//	//If Soft EStop is pressed, turn off 1027, 1028, 1029, 1030, 1031
//	IF KR4_Estop THEN		
//		bOutBit[2,0]:=bOutBit[2,1]:=bOutBit[2,2]:=bOutBit[2,3]:=bOutBit[2,4]:=bOutBit[2,5]:=bOutBit[2,6]:=FALSE;
//	END_IF
	
//	//================================ Function IO
	
//	PLC_O_D2.0 := bOutBit[2,0]; //1027
//	PLC_O_D2.1 := bOutBit[2,1]; //1028
//	PLC_O_D2.2 := bOutBit[2,2]; //1029
//	PLC_O_D2.3 := bOutBit[2,3]; //1030
//	PLC_O_D2.4 := bOutBit[2,4]; //1031
//	PLC_O_D2.5 := bOutBit[2,5]; //1032
//	PLC_O_D2.6 := bOutBit[2,6]; //1033
//	PLC_O_D2.7 := bOutBit[2,7]; //1034
	
//	PLC_O_D3.0 := bOutBit[3,0]; //1035
//	PLC_O_D3.1 := bOutBit[3,1]; //1036
//	PLC_O_D3.2 := bOutBit[3,2]; //1037
//	PLC_O_D3.3 := bOutBit[3,3]; //1038
//	PLC_O_D3.4 := bOutBit[3,4]; //1039
//	PLC_O_D3.5 := bOutBit[3,5]; //1040
//	PLC_O_D3.6 := bOutBit[3,6]; //1041
//	PLC_O_D3.7 := bOutBit[3,7]; //1042
	
//	bInBit[2,0] := PLC_I_D2.0; //993
//	bInBit[2,1] := PLC_I_D2.1; //994
//	bInBit[2,2] := PLC_I_D2.2; //995
//	bInBit[2,3] := PLC_I_D2.3; //996
//	bInBit[2,4] := PLC_I_D2.4; //997
//	bInBit[2,5] := PLC_I_D2.5; //998
//	bInBit[2,6] := PLC_I_D2.6; //999
//	bInBit[2,7] := PLC_I_D2.7; //1000
	
//	bInBit[3,0] := PLC_I_D3.0; //1001
//	bInBit[3,1] := PLC_I_D3.1; //1002
//	bInBit[3,2] := PLC_I_D3.2; //1003
//	bInBit[3,3] := PLC_I_D3.3; //1004
//	bInBit[3,4] := PLC_I_D3.4; //1005
//	bInBit[3,5] := PLC_I_D3.5; //1006
//	bInBit[3,6] := PLC_I_D3.6; //1007
//	bInBit[3,7] := PLC_I_D3.7; //1008

//	//================================ Motion IO
	
//	IF NoMotion THEN
//		RETURN;
//	END_IF
	
//	PLC_O_D1.0 := bOutBit[1,0]; //300
//	PLC_O_D1.1 := bOutBit[1,1]; //301
//	PLC_O_D1.2 := bOutBit[1,2]; //302
//	PLC_O_D1.3 := bOutBit[1,3]; //303
//	PLC_O_D1.4 := bOutBit[1,4]; //304
//	PLC_O_D1.5 := bOutBit[1,5]; //305
//	PLC_O_D1.6 := bOutBit[1,6]; //306
//	PLC_O_D1.7 := bOutBit[1,7]; //307
	
//	bInBit[1,0] := PLC_I_D1.0; //300
//	bInBit[1,1] := PLC_I_D1.1; //301
//	bInBit[1,2] := PLC_I_D1.2; //302
//	bInBit[1,3] := PLC_I_D1.3; //303
//	bInBit[1,4] := PLC_I_D1.4; //304
//	bInBit[1,5] := PLC_I_D1.5; //305
//	bInBit[1,6] := PLC_I_D1.6; //306
//	bInBit[1,7] := PLC_I_D1.7; //307
	
//	IF PLC_I_D1 = 1 THEN
//		Idle := TRUE;
//	ELSE
//		Idle := FALSE;
//	END_IF

END_PROGRAM

// ---- POUs/Kuka IO/KR5.TcPOU
PROGRAM KR5
VAR_INPUT
	PLC_O_SYS 	AT %Q* : DWORD;
	PLC_O_PROG1 AT %Q* : DWORD;
	
	PLC_I_SYS 	AT %I* : DWORD;
	PLC_I_PROG1 AT %I* : DWORD;
	PLC_I_AXIS 	AT %I* : ARRAY[1..6] OF DWORD;
	PLC_I_CURR	AT %I* : ARRAY[1..6] OF DWORD;
	PLC_I_TEMP	AT %I* : ARRAY[1..6] OF DWORD;
	
	KR5_Estop		: BOOL;
	Idle			: BOOL;
	NoMotion		: BOOL;
	
	bOutBit : ARRAY [1..6,0..7] OF BOOL;
	bInBit  : ARRAY [1..6,0..7] OF BOOL;
	index		: USINT;
	index1		: USINT;
	
	dAxis		: ARRAY[1..6] OF DWORD;
	dCurr		: ARRAY[1..6] OF DWORD;
	dTemp		: ARRAY[1..6] OF DWORD;
END_VAR

VAR
	KROnline: BOOL;
	KR_ProgReady: BOOL;
END_VAR

	//If Soft EStop is pressed, turn off 1027 ~ 1034
	IF KR5_Estop THEN		
		bOutBit[1,0]:=bOutBit[1,1]:=bOutBit[1,2]:=bOutBit[1,3]:=
		bOutBit[1,4]:=bOutBit[1,5]:=bOutBit[1,6]:=bOutBit[1,7]:=FALSE;
	END_IF

	//Idle 	
	IF 	PLC_I_PROG1 = 1 THEN
			Idle := TRUE;
	ELSE
			Idle := FALSE;	
	END_IF
	
	//Online
	IF bInBit[1,0] OR bInBit[1,3] THEN
		KROnline := TRUE;
	ELSE
		KROnline := FALSE;
	END_IF

	//Program Ready
	IF bInBit[1,6] AND bInBit[2,4] THEN
		KR_ProgReady := TRUE;
	ELSIF GVL.KR1_bypass THEN
		KR_ProgReady := TRUE;
	ELSE
		KR_ProgReady := FALSE;
	END_IF
	
	
	// ======================================================================== System IO
	// Data In
	FOR index := 0 TO 31 BY 1 DO
		IF index < 8 THEN
			bInBit[1,index] := DWORD_TO_BOOL( SHR(PLC_I_SYS,index) AND 1);
		ELSIF index > 7 AND index < 16 THEN
			bInBit[2,index-8] := DWORD_TO_BOOL( SHR(PLC_I_SYS,index) AND 1);
		END_IF
	END_FOR
	
	// Data Out
	PLC_O_SYS.0 := bOutBit[1,0]; // 1027 move_enable
	PLC_O_SYS.1 := bOutBit[1,1]; // 1028 Drive_off
	PLC_O_SYS.2 := bOutBit[1,2]; // 1029 IO_Activate
	PLC_O_SYS.3 := bOutBit[1,3]; // 1030 Ext_Start
	PLC_O_SYS.4 := bOutBit[1,4]; // 1031 Conf_mess
	PLC_O_SYS.5 := bOutBit[1,5]; // 1032 
	PLC_O_SYS.6 := bOutBit[1,6]; // 1033 Drive_on
	PLC_O_SYS.7 := bOutBit[1,7]; // 1034 Pgno_Fbit
	PLC_O_SYS.8 := bOutBit[2,0]; // 1035 Pgno_Valid
	PLC_O_SYS.9 := bOutBit[2,1]; // 1036 Pgno_Parity

	// ===================================================================== Programme IO
	FOR index := 0 TO 31 BY 1 DO
		IF index < 8 THEN
			bInBit[3,index] := DWORD_TO_BOOL( SHR(PLC_I_PROG1,index) AND 1);
		ELSIF index > 7 AND index < 16 THEN
			bInBit[4,index-8] := DWORD_TO_BOOL( SHR(PLC_I_PROG1,index) AND 1);
		ELSIF index > 15 AND index < 24 THEN
			bInBit[5,index-16] := DWORD_TO_BOOL( SHR(PLC_I_PROG1,index) AND 1);
		ELSIF index > 23 THEN
			bInBit[6,index-24] := DWORD_TO_BOOL( SHR(PLC_I_PROG1,index) AND 1);
		END_IF
	END_FOR
	
	
	PLC_O_PROG1.0 := bOutBit[3,0]; // 200
	PLC_O_PROG1.1 := bOutBit[3,1]; // 201
	PLC_O_PROG1.2 := bOutBit[3,2]; // 202
	PLC_O_PROG1.3 := bOutBit[3,3]; // 203
	PLC_O_PROG1.4 := bOutBit[3,4]; // 204
	PLC_O_PROG1.5 := bOutBit[3,5]; // 205
	PLC_O_PROG1.6 := bOutBit[3,6]; // 206
	PLC_O_PROG1.7 := bOutBit[3,7]; // 207
	PLC_O_PROG1.8 := bOutBit[4,0]; // 208
	PLC_O_PROG1.9 := bOutBit[4,1]; // 209
	PLC_O_PROG1.10 := bOutBit[4,2]; // 210
	PLC_O_PROG1.11 := bOutBit[4,3]; // 211
	PLC_O_PROG1.12 := bOutBit[4,4]; // 212
	PLC_O_PROG1.13 := bOutBit[4,5]; // 213
	PLC_O_PROG1.14 := bOutBit[4,6]; // 214
	PLC_O_PROG1.15 := bOutBit[4,7]; // 215
	PLC_O_PROG1.16 := bOutBit[5,0]; // 216
	PLC_O_PROG1.17 := bOutBit[5,1]; // 217
	PLC_O_PROG1.18 := bOutBit[5,2]; // 218
	PLC_O_PROG1.19 := bOutBit[5,3]; // 219
	PLC_O_PROG1.20 := bOutBit[5,4]; // 220
	PLC_O_PROG1.21 := bOutBit[5,5]; // 221
	PLC_O_PROG1.22 := bOutBit[5,6]; // 222
	PLC_O_PROG1.23 := bOutBit[5,7]; // 223
	PLC_O_PROG1.24 := bOutBit[6,0]; // 224
	PLC_O_PROG1.25 := bOutBit[6,1]; // 225
	PLC_O_PROG1.26 := bOutBit[6,2]; // 226
	PLC_O_PROG1.27 := bOutBit[6,3]; // 227
	PLC_O_PROG1.28 := bOutBit[6,4]; // 228
	PLC_O_PROG1.29 := bOutBit[6,5]; // 229
	PLC_O_PROG1.30 := bOutBit[6,6]; // 230
	PLC_O_PROG1.31 := bOutBit[6,7]; // 231
	
	// ===================================================================== Robot Data
	FOR index1 := 1 TO 6 BY 1 DO
		FOR index := 0 TO 31 BY 1 DO
			dAxis[index1] := PLC_I_AXIS[index1];
			dCurr[index1] := PLC_I_CURR[index1];
			dTemp[index1] := PLC_I_TEMP[index1];
		END_FOR
	END_FOR
	
	
	
	
	
	
	
	
	
//	//================================ Function IO
	
//	PLC_O_D1.0 := bOutBit[1,0]; //1027 motion enable (on to start motor)
//	PLC_O_D1.1 := bOutBit[1,1]; //1028 Drives off (inverse) (on to start motor)
//	PLC_O_D1.2 := bOutBit[1,2]; //1029 Activate interface (on to start motor)
//	PLC_O_D1.3 := bOutBit[1,3]; //1030 Prog Start
//	PLC_O_D1.4 := bOutBit[1,4]; //1031 Acknowledge error msg
//	PLC_O_D1.5 := bOutBit[1,5]; //1032 Drives on
//	PLC_O_D1.6 := bOutBit[1,6]; //1033
//	PLC_O_D1.7 := bOutBit[1,7]; //1034
	
//	PLC_O_D2.0 := bOutBit[2,0]; //1035
//	PLC_O_D2.1 := bOutBit[2,1]; //1036
//	PLC_O_D2.2 := bOutBit[2,2]; //1037
//	PLC_O_D2.3 := bOutBit[2,3]; //1038
//	PLC_O_D2.4 := bOutBit[2,4]; //1039
//	PLC_O_D2.5 := bOutBit[2,5]; //1040
//	PLC_O_D2.6 := bOutBit[2,6]; //1041
//	PLC_O_D2.7 := bOutBit[2,7]; //1042
	
//	bInBit[1,0] := PLC_I_D1.0; //993
//	bInBit[1,1] := PLC_I_D1.1; //994
//	bInBit[1,2] := PLC_I_D1.2; //995
//	bInBit[1,3] := PLC_I_D1.3; //996
//	bInBit[1,4] := PLC_I_D1.4; //997
//	bInBit[1,5] := PLC_I_D1.5; //998
//	bInBit[1,6] := PLC_I_D1.6; //999
//	bInBit[1,7] := PLC_I_D1.7; //1000
	
//	bInBit[2,0] := PLC_I_D2.0; //1001
//	bInBit[2,1] := PLC_I_D2.1; //1002
//	bInBit[2,2] := PLC_I_D2.2; //1003
//	bInBit[2,3] := PLC_I_D2.3; //1004
//	bInBit[2,4] := PLC_I_D2.4; //1005
//	bInBit[2,5] := PLC_I_D2.5; //1006
//	bInBit[2,6] := PLC_I_D2.6; //1007
//	bInBit[2,7] := PLC_I_D2.7; //1008
	
//	//================================ Motion IO
	
//	IF NoMotion THEN
//		RETURN;
//	END_IF
	
//	PLC_O_D3.0 := bOutBit[3,0]; //200
//	PLC_O_D3.1 := bOutBit[3,1]; //201
//	PLC_O_D3.2 := bOutBit[3,2]; //202
//	PLC_O_D3.3 := bOutBit[3,3]; //203
//	PLC_O_D3.4 := bOutBit[3,4]; //204
//	PLC_O_D3.5 := bOutBit[3,5]; //205
//	PLC_O_D3.6 := bOutBit[3,6]; //206
//	PLC_O_D3.7 := bOutBit[3,7]; //207
	
//	PLC_O_D4.0 := bOutBit[4,0]; //208
//	PLC_O_D4.1 := bOutBit[4,1]; //209
//	PLC_O_D4.2 := bOutBit[4,2]; //210
//	PLC_O_D4.3 := bOutBit[4,3]; //211
//	PLC_O_D4.4 := bOutBit[4,4]; //212
//	PLC_O_D4.5 := bOutBit[4,5]; //213
//	PLC_O_D4.6 := bOutBit[4,6]; //214
//	PLC_O_D4.7 := bOutBit[4,7]; //215
	
//	PLC_O_D5.0 := bOutBit[5,0]; //216
//	PLC_O_D5.1 := bOutBit[5,1]; //217
//	PLC_O_D5.2 := bOutBit[5,2]; //218
//	PLC_O_D5.3 := bOutBit[5,3]; //219
//	PLC_O_D5.4 := bOutBit[5,4]; //220
//	PLC_O_D5.5 := bOutBit[5,5]; //221
//	PLC_O_D5.6 := bOutBit[5,6]; //222
//	PLC_O_D5.7 := bOutBit[5,7]; //223

//	PLC_O_D6.0 := bOutBit[6,0]; //224
//	PLC_O_D6.1 := bOutBit[6,1]; //225
//	PLC_O_D6.2 := bOutBit[6,2]; //226
//	PLC_O_D6.3 := bOutBit[6,3]; //227
//	PLC_O_D6.4 := bOutBit[6,4]; //228
//	PLC_O_D6.5 := bOutBit[6,5]; //229
//	PLC_O_D6.6 := bOutBit[6,6]; //230
//	PLC_O_D6.7 := bOutBit[6,7]; //231

//	bInBit[3,0] := PLC_I_D3.0; //200
//	bInBit[3,1] := PLC_I_D3.1; //201
//	bInBit[3,2] := PLC_I_D3.2; //202
//	bInBit[3,3] := PLC_I_D3.3; //203
//	bInBit[3,4] := PLC_I_D3.4; //204
//	bInBit[3,5] := PLC_I_D3.5; //205
//	bInBit[3,6] := PLC_I_D3.6; //206
//	bInBit[3,7] := PLC_I_D3.7; //207
	
//	bInBit[4,0] := PLC_I_D4.0; //208
//	bInBit[4,1] := PLC_I_D4.1; //209
//	bInBit[4,2] := PLC_I_D4.2; //210
//	bInBit[4,3] := PLC_I_D4.3; //211
//	bInBit[4,4] := PLC_I_D4.4; //212
//	bInBit[4,5] := PLC_I_D4.5; //213
//	bInBit[4,6] := PLC_I_D4.6; //214
//	bInBit[4,7] := PLC_I_D4.7; //215
	
//	bInBit[5,0] := PLC_I_D5.0; //216
//	bInBit[5,1] := PLC_I_D5.1; //217
//	bInBit[5,2] := PLC_I_D5.2; //218
//	bInBit[5,3] := PLC_I_D5.3; //219
//	bInBit[5,4] := PLC_I_D5.4; //220
//	bInBit[5,5] := PLC_I_D5.5; //221
//	bInBit[5,6] := PLC_I_D5.6; //222
//	bInBit[5,7] := PLC_I_D5.7; //223
	
//	bInBit[6,0] := PLC_I_D6.0; //224
//	bInBit[6,1] := PLC_I_D6.1; //225
//	bInBit[6,2] := PLC_I_D6.2; //226
//	bInBit[6,3] := PLC_I_D6.3; //227
//	bInBit[6,4] := PLC_I_D6.4; //228
//	bInBit[6,5] := PLC_I_D6.5; //229
//	bInBit[6,6] := PLC_I_D6.6; //230
//	bInBit[6,7] := PLC_I_D6.7; //231
	
	
	
//	//If Soft EStop is pressed, turn off 1027, 1028, 1029, 1030, 1031
//	IF KR5_Estop THEN		
//		bOutBit[3,0]:=bOutBit[3,1]:=bOutBit[3,2]:=bOutBit[3,3]:=bOutBit[3,4]:=bOutBit[2,5]:=bOutBit[2,6]:=FALSE;
//	END_IF
	
//	//================================ Function IO
	
//	PLC_O_D3.0 := bOutBit[3,0]; //1027
//	PLC_O_D3.1 := bOutBit[3,1]; //1028
//	PLC_O_D3.2 := bOutBit[3,2]; //1029
//	PLC_O_D3.3 := bOutBit[3,3]; //1030
//	PLC_O_D3.4 := bOutBit[3,4]; //1031
//	PLC_O_D3.5 := bOutBit[3,5]; //1032
//	PLC_O_D3.6 := bOutBit[3,6]; //1033
//	PLC_O_D3.7 := bOutBit[3,7]; //1034
	
//	PLC_O_D4.0 := bOutBit[4,0]; //1035
//	PLC_O_D4.1 := bOutBit[4,1]; //1036
//	PLC_O_D4.2 := bOutBit[4,2]; //1037
//	PLC_O_D4.3 := bOutBit[4,3]; //1038
//	PLC_O_D4.4 := bOutBit[4,4]; //1039
//	PLC_O_D4.5 := bOutBit[4,5]; //1040
//	PLC_O_D4.6 := bOutBit[4,6]; //1041
//	PLC_O_D4.7 := bOutBit[4,7]; //1042
	
//	bInBit[3,0] := PLC_I_D3.0; //993
//	bInBit[3,1] := PLC_I_D3.1; //994
//	bInBit[3,2] := PLC_I_D3.2; //995
//	bInBit[3,3] := PLC_I_D3.3; //996
//	bInBit[3,4] := PLC_I_D3.4; //997
//	bInBit[3,5] := PLC_I_D3.5; //998
//	bInBit[3,6] := PLC_I_D3.6; //999
//	bInBit[3,7] := PLC_I_D3.7; //1000
	
//	bInBit[4,0] := PLC_I_D4.0; //1001
//	bInBit[4,1] := PLC_I_D4.1; //1002
//	bInBit[4,2] := PLC_I_D4.2; //1003
//	bInBit[4,3] := PLC_I_D4.3; //1004
//	bInBit[4,4] := PLC_I_D4.4; //1005
//	bInBit[4,5] := PLC_I_D4.5; //1006
//	bInBit[4,6] := PLC_I_D4.6; //1007
//	bInBit[4,7] := PLC_I_D4.7; //1008
	
//	//================================ Motion IO
	
//	IF NoMotion THEN
//		RETURN;
//	END_IF

//	PLC_O_D1.0 := bOutBit[1,0]; //200
//	PLC_O_D1.1 := bOutBit[1,1]; //201
//	PLC_O_D1.2 := bOutBit[1,2]; //202
//	PLC_O_D1.3 := bOutBit[1,3]; //203
//	PLC_O_D1.4 := bOutBit[1,4]; //204
//	PLC_O_D1.5 := bOutBit[1,5]; //205
//	PLC_O_D1.6 := bOutBit[1,6]; //206
//	PLC_O_D1.7 := bOutBit[1,7]; //207
	
//	PLC_O_D2.0 := bOutBit[2,0]; //208
//	PLC_O_D2.1 := bOutBit[2,1]; //209
//	PLC_O_D2.2 := bOutBit[2,2]; //210
//	PLC_O_D2.3 := bOutBit[2,3]; //211
//	PLC_O_D2.4 := bOutBit[2,4]; //212
//	PLC_O_D2.5 := bOutBit[2,5]; //213
//	PLC_O_D2.6 := bOutBit[2,6]; //214
//	PLC_O_D2.7 := bOutBit[2,7]; //215
	
//	bInBit[1,0] := PLC_I_D1.0; //200
//	bInBit[1,1] := PLC_I_D1.1; //201
//	bInBit[1,2] := PLC_I_D1.2; //202
//	bInBit[1,3] := PLC_I_D1.3; //203
//	bInBit[1,4] := PLC_I_D1.4; //204
//	bInBit[1,5] := PLC_I_D1.5; //205
//	bInBit[1,6] := PLC_I_D1.6; //206
//	bInBit[1,7] := PLC_I_D1.7; //207
	
//	bInBit[2,0] := PLC_I_D2.0; //208
//	bInBit[2,1] := PLC_I_D2.1; //209
//	bInBit[2,2] := PLC_I_D2.2; //210
//	bInBit[2,3] := PLC_I_D2.3; //211
//	bInBit[2,4] := PLC_I_D2.4; //212
//	bInBit[2,5] := PLC_I_D2.5; //213
//	bInBit[2,6] := PLC_I_D2.6; //214
//	bInBit[2,7] := PLC_I_D2.7; //215

//	IF PLC_I_D1 = 1 THEN
//		Idle := TRUE;
//	ELSE
//		Idle := FALSE;
//	END_IF

END_PROGRAM

// ---- POUs/RESET_SEQ.TcPOU
PROGRAM RESET_SEQ
VAR_INPUT
	Reset_seq	: INT;
	log_reset	: STRING[255];
END_VAR
VAR
	RstTON		: TON;
	RstToff		: TON;
	bOn			: BOOL;
	bLastOn		: BOOL;
	Bit1		: INT;
	Bit2		: INT;
END_VAR


	//Off time
	RstTON(IN:= NOT RstTOff.Q, PT:= T#0.2S, Q=> bOn , ET=> );
	//On time
	RstTOff(IN:= bOn, PT:= T#0.5S, Q=> , ET=> );
	
	IF bOn <> bLastOn THEN
		IF bON THEN
			IF Reset_seq < 14 THEN
				IF Reset_seq =2 THEN
					IF KR1.bInBit[1,6] AND KR2.bInBit[1,6] AND KR3.bInBit[1,6] AND KR4.bInBit[1,6] AND KR5.bInBit[1,6] THEN
						Reset_seq := Reset_seq + 1;	
					END_IF
				ELSE	
					Reset_seq := Reset_seq + 1;
				END_IF			
			ELSE
				Reset_seq 	:=0;
				bOn 		:= FALSE;
			END_IF
		END_IF
	END_IF
	
	CASE Reset_seq OF
		0:
			IF NOT GVL.KR1_bypass THEN
				FOR Bit1 := 1 TO 30 BY 1 DO
					FOR Bit2 := 0 TO 7 BY 1 DO
						KR1.bOutBit[Bit1,Bit2] := FALSE;
					END_FOR
				END_FOR
			END_IF
			IF NOT GVL.KR2_bypass THEN
				FOR Bit1 := 1 TO 8 BY 1 DO
					FOR Bit2 := 0 TO 7 BY 1 DO
						KR2.bOutBit[Bit1,Bit2] := FALSE;
					END_FOR
				END_FOR
			END_IF
			IF NOT GVL.KR3_bypass THEN
				FOR Bit1 := 1 TO 3 BY 1 DO
					FOR Bit2 := 0 TO 7 BY 1 DO
						KR3.bOutBit[Bit1,Bit2] := FALSE;
					END_FOR
				END_FOR
			END_IF
			IF NOT GVL.KR4_bypass THEN
				FOR Bit1 := 1 TO 3 BY 1 DO
					FOR Bit2 := 0 TO 7 BY 1 DO
						KR4.bOutBit[Bit1,Bit2] := FALSE;
					END_FOR
				END_FOR
			END_IF
			IF NOT GVL.KR5_bypass THEN
				FOR Bit1 := 1 TO 6 BY 1 DO
					FOR Bit2 := 0 TO 7 BY 1 DO
						KR5.bOutBit[Bit1,Bit2] := FALSE;
					END_FOR
				END_FOR
			END_IF
		1:
			IF NOT GVL.KR1_bypass THEN
				KR1.bOutBit[1,0]:=KR1.bOutBit[1,1]:=KR1.bOutBit[1,2]:=TRUE;
			END_IF
			IF NOT GVL.KR2_bypass THEN
				KR2.bOutBit[1,0]:=KR2.bOutBit[1,1]:=KR2.bOutBit[1,2]:=TRUE;
			END_IF
			IF NOT GVL.KR3_bypass THEN
				KR3.bOutBit[1,0]:=KR3.bOutBit[1,1]:=KR3.bOutBit[1,2]:=TRUE;
			END_IF
			IF NOT GVL.KR4_bypass THEN
				KR4.bOutBit[1,0]:=KR4.bOutBit[1,1]:=KR4.bOutBit[1,2]:=TRUE;
			END_IF
			IF NOT GVL.KR5_bypass THEN
				KR5.bOutBit[1,0]:=KR5.bOutBit[1,1]:=KR5.bOutBit[1,2]:=TRUE;
			END_IF
		2:
			IF NOT GVL.KR1_bypass THEN
				KR1.bOutBit[1,4] := TRUE; //1031
			END_IF
			IF NOT GVL.KR2_bypass THEN
				KR2.bOutBit[1,4] := TRUE; //1031
			END_IF
			IF NOT GVL.KR3_bypass THEN
				KR3.bOutBit[1,4] := TRUE; //1031
			END_IF
			IF NOT GVL.KR4_bypass THEN
				KR4.bOutBit[1,4] := TRUE; //1031
			END_IF
			IF NOT GVL.KR5_bypass THEN
				KR5.bOutBit[1,4] := TRUE; //1031
			END_IF
		3:
			IF NOT GVL.KR1_bypass THEN
				KR1.bOutBit[1,4] := FALSE; //1031
			END_IF
			IF NOT GVL.KR2_bypass THEN
				KR2.bOutBit[1,4] := FALSE; //1031
			END_IF
			IF NOT GVL.KR3_bypass THEN
				KR3.bOutBit[1,4] := FALSE; //1031
			END_IF
			IF NOT GVL.KR4_bypass THEN
				KR4.bOutBit[1,4] := FALSE; //1031
			END_IF
			IF NOT GVL.KR5_bypass THEN
				KR5.bOutBit[1,4] := FALSE; //1031
			END_IF
		4:
			KR1.bOutBit[1,5] := TRUE; //1032
		5:
			KR2.bOutBit[1,6] := TRUE; //1033
		6:
			KR3.bOutBit[1,5] := TRUE; //1032
		7:	
			KR4.bOutBit[1,5] := TRUE; //1032
		8:		
			KR5.bOutBit[1,5] := TRUE; //1032
		9:
			KR1.bOutBit[1,5] := FALSE; //1032
			KR1.bOutBit[1,3] := TRUE; //1030
		10:
			KR2.bOutBit[1,6] := FALSE; //1033
			KR2.bOutBit[1,3] := TRUE; //1030
		11:
			KR3.bOutBit[1,5] := FALSE; //1032
			KR3.bOutBit[1,3] := TRUE; //1030
		12:
			KR4.bOutBit[1,5] := FALSE; //1032
			KR4.bOutBit[1,3] := TRUE; //1030
		13:
			KR5.bOutBit[1,5] := FALSE; //1032
			KR5.bOutBit[1,3] := TRUE; //1030
		14:
			AUTO_MODE.Halt_Production := FALSE;
			Reset_seq :=0;
			MAIN.Reset_State := FALSE;
			MAIN.btn_Reset := FALSE;
	END_CASE
	bLastOn := bOn;

END_PROGRAM

// ---- POUs/Auto_Seq/AUTO_MODE.TcPOU
PROGRAM AUTO_MODE
VAR_INPUT
	Reset_seq_btn	: BOOL;
	Start_time	: string;
	
	JIGA_WELDING: BOOL;
	JIGB_WELDING: BOOL;
	JIGC_WELDING: BOOL;
	TT_WELDING	: BOOL;
	IF_PICK		: BOOL;
	JIGC_PICK	: BOOL;
	VB_PICK		: BOOL;
	
	JIGA_LOAD	: BOOL;
	JIGB_LOAD	: BOOL;
	JIGC_LOAD	: BOOL;
	TT_LOAD		: BOOL;
	CR_PICK		: BOOL;
	
	AutoMode	: BOOL;
	ManualMode	: BOOL;
	next_step	: BOOL;
	Halt_Production	: BOOL;
	
	processnameA5 : STRING[255];
	processnameA4 : STRING[255];
	processnameA3 : STRING[255];
	processnameA2 : STRING[255];
	processnameA1 : STRING[255];
	processnameCR : STRING[255];
	processnameRW : STRING[255];
	processnameFG : STRING[255];
	processnameCOSMO : STRING[255];
	
	COSMO_LOAD	: BOOL;
	COSMO_RUN	: BOOL;
	CR_UNLOADING: BOOL;
	
	CLEAR_COSMO	: Bool;
	KR1_PITSTOP : BOOL;
	FG_PACKING	: BOOL;
	RW_PACKING	: BOOL;
	
	A4_Run_Flag : BOOL;
	A3_Run_Flag : BOOL;
	A2_Run_Flag : BOOL;
	A1_Run_Flag : BOOL;
	
	Run_Next_Rack : BOOL:= TRUE;
	Out_time	: STRING;
	JIGA_ErrorState : BOOL;
	JIGB_ErrorState : BOOL;
	JIGC_ErrorState : BOOL;
	TT_ErrorState 	: BOOL;
END_VAR
VAR
	Auto_IntOn	: TON;
	Auto_IntOff	: TON;
	Auto_on		: BOOL;
	Auto_laston	: BOOL;
	
	Bit1: INT;
	Bit2: INT;
END_VAR

IF next_step OR Automode THEN
	IF NOT KR2.KR_ProgReady OR NOT KR3.KR_ProgReady OR NOT KR4.KR_ProgReady OR NOT KR5.KR_ProgReady THEN
		Automode := FALSE;
	END_IF
	IF_RACK_CHECK();
	SEQ_A5();
	SEQ_A4();
	SEQ_A3();
	SEQ_A2();
	SEQ_A1();
	SEQ_B5();
	SEQ_B4();
	SEQ_B3();
	SEQ_B2();
	SEQ_B1();
		
	SEQ_CR_PICK();
//	SEQ_LP_LYR0();
	SEQ_FG_A();
	SEQ_COSMO();
	
	 
END_IF




IF Reset_seq_btn THEN
	
	
	IF_RACK_CHECK.checkIn_A5 := IF_RACK_CHECK.checkIn_A4 := IF_RACK_CHECK.checkIn_A3 := IF_RACK_CHECK.checkIn_A2 := IF_RACK_CHECK.checkIn_A1 := 
	IF_RACK_CHECK.checkIn_B5 := IF_RACK_CHECK.checkIn_B4 := IF_RACK_CHECK.checkIn_B3 := IF_RACK_CHECK.checkIn_B2 := IF_RACK_CHECK.checkIn_B1 := FALSE;
	
	SEQ_A5.A5_sequence		:= SEQ_A4.A4_sequence		:= SEQ_A3.A3_sequence	:= SEQ_A2.A2_sequence	:= SEQ_A1.A1_sequence:=
	SEQ_B5.B5_sequence		:= SEQ_B4.B4_sequence		:= SEQ_B3.B3_sequence	:= SEQ_B2.B2_sequence	:= SEQ_B1.B1_sequence:=
	SEQ_CR_PICK.CR_sequence	:= SEQ_COSMO.COSMO_sequence	:= SEQ_RW.RW_sequence 	:= SEQ_FG_A.FG_sequence	:= SEQ_LYR_PD0.LYRPD_sequence := 0;
	
	processnameA5 := processnameA4 := processnameA3 := processnameA2 	:= processnameA1 :=
	processnameCR := processnameRW := processnameFG := processnameCOSMO := '';  
	
	IF_PICK			:= JIGC_PICK		:= CR_PICK			:=
	JIGA_WELDING 	:= JIGB_WELDING 	:= JIGC_WELDING		:= TT_WELDING   	:= 
	JIGA_LOAD 	 	:= JIGB_LOAD  	 	:= JIGC_LOAD 		:= TT_LOAD			:=
	GVL.JIGA_Clamp 	:= GVL.JIGB_Clamp 	:= GVL.JIGC_Clamp 	:= CR_UNLOADING	 	:= 
	COSMO_LOAD 	 	:= COSMO_RUN 	 	:= CLEAR_COSMO  	:= KR1_PITSTOP 		:= 
	FG_PACKING 	 	:= RW_PACKING 		:= GVL.COSMO_Run	:= GVL.TTorch_Run 	:= FALSE;
	
	JIGA_ErrorState := JIGB_ErrorState 	:= JIGC_ErrorState 	:= TT_ErrorState 	:= FALSE;
	Automode 		:= next_step 		:= FALSE;
	Run_Next_Rack 	:= TRUE;
	Halt_Production := FALSE;
	
	GVL.Layerpad := FALSE;
	GVL.COSMO_UNLOAD := FALSE;

	FOR Bit1 := 2 TO 30 BY 1 DO
		FOR Bit2 := 0 TO 7 BY 1 DO
			KR1.bOutBit[Bit1,Bit2] := FALSE;
		END_FOR
	END_FOR
	FOR Bit1 := 2 TO 8 BY 1 DO
		FOR Bit2 := 0 TO 7 BY 1 DO
			KR2.bOutBit[Bit1,Bit2] := FALSE;
		END_FOR
	END_FOR
	FOR Bit1 := 2 TO 3 BY 1 DO
		FOR Bit2 := 0 TO 7 BY 1 DO
			KR3.bOutBit[Bit1,Bit2] := FALSE;
			KR4.bOutBit[Bit1,Bit2] := FALSE;
		END_FOR
	END_FOR
	FOR Bit1 := 2 TO 6 BY 1 DO
		FOR Bit2 := 0 TO 7 BY 1 DO
			KR5.bOutBit[Bit1,Bit2] := FALSE;
		END_FOR
	END_FOR
	
	Reset_seq_btn := False;
END_IF

END_PROGRAM

// ---- POUs/Auto_Seq/IF_RACK_CHECK.TcPOU
PROGRAM IF_RACK_CHECK
VAR_INPUT
	checkIn_A5 : BOOL;
	checkIn_A4 : BOOL;
	checkIn_A3 : BOOL;
	checkIn_A2 : BOOL;
	checkIn_A1 : BOOL;
	checkIn_B5 : BOOL;
	checkIn_B4 : BOOL;
	checkIn_B3 : BOOL;
	checkIn_B2 : BOOL;
	checkIn_B1 : BOOL;
END_VAR
VAR
	infeedRack_A_empty: BOOL;
	infeedRack_B_empty: BOOL;
	turnflag: BOOL;
	turningA: BOOL;
	turningB: BOOL;
	cool_rack_check : UINT;
END_VAR


IF NOT AUTO_MODE.Run_Next_Rack THEN
	RETURN;
END_IF
	
IF COOL_RACK.CR_full THEN
	RETURN;
END_IF

IF INFEED_RACK.FaceA_InWC THEN
	IF INFEED_RACK.A5_Sensor THEN
		checkIn_A5 := TRUE; AUTO_MODE.Run_Next_Rack := FALSE;
	ELSIF INFEED_RACK.A4_Sensor THEN
		checkIn_A4 := TRUE; AUTO_MODE.Run_Next_Rack := FALSE;
	ELSIF INFEED_RACK.A3_Sensor THEN
		checkIn_A3 := TRUE; AUTO_MODE.Run_Next_Rack := FALSE;
	ELSIF INFEED_RACK.A2_Sensor THEN
		checkIn_A2 := TRUE; AUTO_MODE.Run_Next_Rack := FALSE;
	ELSIF INFEED_RACK.A1_Sensor THEN
		checkIn_A1 := TRUE; AUTO_MODE.Run_Next_Rack := FALSE;
	ELSE
		infeedRack_A_empty := TRUE;	
	END_IF
	
ELSIF INFEED_RACK.FaceB_InWC THEN
	IF INFEED_RACK.B5_Sensor THEN
		checkIn_B5 := TRUE; AUTO_MODE.Run_Next_Rack := FALSE;
	ELSIF INFEED_RACK.B4_Sensor THEN
		checkIn_B4 := TRUE; AUTO_MODE.Run_Next_Rack := FALSE;
	ELSIF INFEED_RACK.B3_Sensor THEN
		checkIn_B3 := TRUE; AUTO_MODE.Run_Next_Rack := FALSE;
	ELSIF INFEED_RACK.B2_Sensor THEN
		checkIn_B2 := TRUE; AUTO_MODE.Run_Next_Rack := FALSE;
	ELSIF INFEED_RACK.B1_Sensor THEN
		checkIn_B1 := TRUE; AUTO_MODE.Run_Next_Rack := FALSE;
	ELSE
		infeedRack_B_empty := TRUE;	
	END_IF
END_IF

IF INFEED_RACK.IFRack_Ready and INFEED_RACK.IFRack_TurnReady THEN
	IF infeedRack_A_empty AND NOT turningB THEN
		turningA := TRUE;
		INFEED_RACK.IFRack_arr[1].5 := FALSE; //BtoA
		INFEED_RACK.IFRack_arr[1].4 := TRUE; //AtoB
		INFEED_RACK(bStart_Write:=TRUE);
		IF INFEED_RACK.FaceB_InWC THEN
			turningA := FALSE;
			infeedRack_A_empty := FALSE;
			INFEED_RACK(bStart_Write:=FALSE);
		END_IF
	ELSIF infeedRack_B_empty AND NOT turningA THEN
		turningB := TRUE;
		INFEED_RACK.IFRack_arr[1].4 := FALSE; //AtoB
		INFEED_RACK.IFRack_arr[1].5 := TRUE; //BtoA
		INFEED_RACK(bStart_Write:=TRUE);
		IF INFEED_RACK.FaceA_InWC THEN
			turningB := FALSE;
			infeedRack_B_empty := FALSE;
			INFEED_RACK(bStart_Write:=FALSE);
		END_IF
	END_IF
END_IF

//INFEED_RACK.bStart_Read:=FALSE;
//INFEED_RACK.bStart_Write:=FALSE;

END_PROGRAM

// ---- POUs/COOL_RACK.TcPOU
PROGRAM COOL_RACK
VAR_INPUT
	bstart_Read		: BOOL;
	bstart_Write	: BOOL;
	iCooling_Time	: INT;
	set_time		: bool;
END_VAR
VAR_OUTPUT
	CR_full 	: bool;
END_VAR
VAR
	WriteCoil	: FB_MBWriteCoils;
	Read_Coils	: FB_MBReadCoils;
	ReadInput: FB_MBReadInputs;
	
	IP_Address		: STRING:='169.254.106.102';
	MB_Port			: UINT	:=502;
	nUnit			: BYTE	:=255; 
	nQuantity		: WORD	:=24;
	nMBAddr			: WORD	:=2048;
	bError_Read		: BOOL;
	bError_Write	: BOOL;
	nErrId_Read		: UDINT;
	nErrId_Write	: UDINT;
	
	CoolRack_arr		: ARRAY [0..2] OF BYTE;

	
	CR	: ARRAY [1..21] OF BOOL;
	num	: INT;
	
	CR_Reset		: INT;
	CR_Sel			: INT;
	CRON			: BOOL;
	CRONlast		: BOOL;
	CRcounterON 	: TON;
	CRcounterOFF	: TON;

END_VAR


//Off time
CRcounterON(IN:= NOT CRcounterOFF.Q, PT:= T#1S, Q=> CRON , ET=> );
//On time
CRcounterOFF(IN:= CRON, PT:= T#1S, Q=> , ET=> );
	
IF CRON <> CRONlast THEN
	FOR CR_Sel := 1 TO 21 BY 1 DO
		IF CR[CR_Sel] THEN
			GVL.CRTimer[CR_Sel] := GVL.CRTimer[CR_Sel] - 1;
		END_IF
	END_FOR
END_IF
CRONlast := CRON;
//================================ Function Block

Read_Coils(
	sIPAddr:= IP_Address, 
	nTCPPort:= MB_Port, 
	nUnitID:= nUnit, 
	nQuantity:= nQuantity, 
	nMBAddr:= nMBAddr, 
	cbLength:= SIZEOF(CoolRack_arr), 
	pDestAddr:= ADR(CoolRack_arr), 
	bExecute:= bstart_Read, 
	tTimeout:= T#1S, 
	bBusy=> , 
	bError=> bError_Read, 
	nErrId=> nErrId_Read, 
	cbRead=> );

WriteCoil(
	sIPAddr:= IP_Address, 
	nTCPPort:= MB_Port, 
	nUnitID:= nUnit, 
	nQuantity:= nQuantity, 
	nMBAddr:= nMBAddr, 
	cbLength:= SIZEOF(CoolRack_arr),  
	pSrcAddr:= ADR(CoolRack_arr), 
	bExecute:= bstart_Write, 
	tTimeout:= T#1S, 
	bBusy=> , 
	bError=> bError_Write, 
	nErrId=> nErrId_Write);

IF set_time THEN
	FOR CR_Reset := 1 TO 21 BY 1 DO
		GVL.CRTimer[CR_Reset] := GVL.iCooling_Time;
	END_FOR	
END_IF

//================================ Sensor

CR[1] := CoolRack_arr[0].0;
CR[2] := CoolRack_arr[0].1;
CR[3] := CoolRack_arr[0].2;
CR[4] := CoolRack_arr[0].3;
CR[5] := CoolRack_arr[0].4;
CR[6] := CoolRack_arr[0].5;
CR[7] := CoolRack_arr[0].6;

CR[8] := CoolRack_arr[0].7;
CR[9] := CoolRack_arr[1].0;
CR[10] := CoolRack_arr[1].1;
CR[11] := CoolRack_arr[1].2;
CR[12] := CoolRack_arr[1].3;
CR[13] := CoolRack_arr[1].4;
CR[14] := CoolRack_arr[1].5;

CR[15] := CoolRack_arr[1].6;
CR[16] := CoolRack_arr[1].7;
CR[17] := CoolRack_arr[2].0;
CR[18] := CoolRack_arr[2].1;
CR[19] := CoolRack_arr[2].2;
CR[20] := CoolRack_arr[2].3;
CR[21] := CoolRack_arr[2].4;

CR[8]:=TRUE;
CR[14]:=TRUE;
CR[15]:=TRUE;
CR[16]:=TRUE;
CR[17]:=TRUE;
CR[18]:=TRUE;
CR[19]:=TRUE;
CR[20]:=TRUE;
CR[21]:=TRUE;
//================================ Cooling Time
FOR num:=1 TO 21 BY 1 DO
	IF NOT CR[num] THEN
		GVL.CRTimer[num] := GVL.iCooling_Time;
	END_IF
//	IF num > 21 THEN
//		num := 1;			
//	END_IF
END_FOR

IF CoolRack_arr[0] = 255 AND CoolRack_arr[1] = 255 AND CoolRack_arr[2] = 31 THEN
	CR_full := TRUE;
ELSE
	CR_full := false;
END_IF

END_PROGRAM

// ---- POUs/INFEED_RACK.TcPOU
PROGRAM INFEED_RACK
VAR_INPUT
	bstart_Read		: BOOL;
	bstart_Write	: BOOL;
	A1_Valve		: BOOL;
	A2_Valve		: BOOL;
	A3_Valve		: BOOL;
	A4_Valve		: BOOL;
	A5_Valve		: BOOL;
	B1_Valve		: BOOL;
	B2_Valve		: BOOL;
	B3_Valve		: BOOL;
	B4_Valve		: BOOL;
	B5_Valve		: BOOL;
	IFRack_Connect	: BOOL;
	IFRack_Ready	: BOOL;
	Turn_A_to_B		: BOOL;
	Turn_B_to_A		: BOOL;
	A1_Sensor		: BOOL;
	A2_Sensor		: BOOL;
	A3_Sensor		: BOOL;
	A4_Sensor		: BOOL;
	A5_Sensor		: BOOL;
	B1_Sensor		: BOOL;
	B2_Sensor		: BOOL;
	B3_Sensor		: BOOL;
	B4_Sensor		: BOOL;
	B5_Sensor		: BOOL;
	FaceA_InWC		: BOOL;
	FaceB_InWC		: BOOL;
	IFRack_TurnReady : BOOL;
	
	IFRack_arr		: ARRAY [0..6] OF BYTE;
END_VAR
VAR
	WriteCoil	: FB_MBWriteCoils;
	Read_Coils	: FB_MBReadCoils;
	ReadInput: FB_MBReadInputs;
	
	IP_Address		: STRING:='169.254.106.101';
	MB_Port			: UINT	:=502;
	nUnit			: BYTE	:=255; 
	nQuantity		: WORD	:=48;
	nMBAddr			: WORD	:=2048;
	bError_Read		: BOOL;
	bError_Write	: BOOL;
	nErrId_Read		: UDINT;
	nErrId_Write	: UDINT;
	
END_VAR


//================================ Function Block

Read_Coils(
	sIPAddr:= IP_Address, 
	nTCPPort:= MB_Port, 
	nUnitID:= nUnit, 
	nQuantity:= nQuantity, 
	nMBAddr:= nMBAddr, 
	cbLength:= SIZEOF(IFRack_arr), 
	pDestAddr:= ADR(IFRack_arr), 
	bExecute:= bstart_Read, 
	tTimeout:= T#1S, 
	bBusy=> , 
	bError=> bError_Read, 
	nErrId=> nErrId_Read, 
	cbRead=> );

WriteCoil(
	sIPAddr:= IP_Address, 
	nTCPPort:= MB_Port, 
	nUnitID:= nUnit, 
	nQuantity:= nQuantity, 
	nMBAddr:= nMBAddr, 
	cbLength:= SIZEOF(IFRack_arr),  
	pSrcAddr:= ADR(IFRack_arr), 
	bExecute:= bstart_Write, 
	tTimeout:= T#1S, 
	bBusy=> , 
	bError=> bError_Write, 
	nErrId=> nErrId_Write);
	
//================================ Sensor

IFRack_arr[0].0	:= A1_Valve;
IFRack_arr[0].1	:= A2_Valve;
IFRack_arr[0].2	:= A3_Valve;
IFRack_arr[0].3	:= A4_Valve;
IFRack_arr[0].4	:= A5_Valve;

IFRack_arr[0].5	:= B1_Valve;
IFRack_arr[0].6	:= B2_Valve;
IFRack_arr[0].7	:= B3_Valve;
IFRack_arr[1].0	:= B4_Valve;
IFRack_arr[1].1	:= B5_Valve;

IFRack_arr[1].2	:= IFRack_Connect;
IFRack_Ready	:= IFRack_arr[1].3;
IFRack_arr[1].4	:= Turn_A_to_B;
IFRack_arr[1].5	:= Turn_B_to_A;

A1_Sensor 		:= IFRack_arr[3].6;
A2_Sensor 		:= IFRack_arr[3].7;
A3_Sensor 		:= IFRack_arr[4].0;
A4_Sensor 		:= IFRack_arr[4].1;
A5_Sensor 		:= IFRack_arr[4].2;

B1_Sensor 		:= IFRack_arr[4].3;
B2_Sensor 		:= IFRack_arr[4].4;
B3_Sensor 		:= IFRack_arr[4].5;
B4_Sensor 		:= IFRack_arr[4].6;
B5_Sensor 		:= IFRack_arr[4].7;

FaceA_InWC		:= IFRack_arr[5].0;
FaceB_InWC		:= IFRack_arr[5].1;
IFRack_TurnReady:= IFRack_arr[5].2;

END_PROGRAM

// ---- POUs/Auto_Seq/SEQ_A5.TcPOU
PROGRAM SEQ_A5
VAR_INPUT
	A5_sequence	: UINT;
	process_A	: UINT; // IF RACK PICK (KR5)
	process_J	: UINT; // PLACE TO JIG A (KR5)
	process_B	: UINT; // JIG A WELDING(KR3)
	process_C	: UINT; // JIG A TO JIG B {KR5}
	process_D	: UINT; // JIG B WELDING (KR3) 
	process_E	: UINT; // JIG B TO TWINTORCH (KR5) 
	process_F	: UINT; // TWINTORCH TO JIG C (KR5)
	process_G	: UINT; // BRACKET TO JIG C (KR2) 
	process_H	: UINT; // JIG C WELDING (KR4)
	process_I	: UINT; // JIG C TO PICK (KR2)
	process_K	: UINT; // PLACE TO CR (KR2)
	
END_VAR
VAR
	Bit1			: INT;
	Bit2			: INT;
	Jig_ErrorTime 	: TIME := T#5S;
	TT_ErrorTime 	: TIME := T#120S;
	JigTimerA 		: TON;
	JigTimerB 		: TON;
	JigTimerC 		: TON;
	TTTimer			: TON;
	Msg_PlaceCR		: STRING;
END_VAR

IF NOT IF_RACK_CHECK.checkIn_A5 
OR NOT INFEED_RACK.IFRack_Ready THEN
	RETURN;
END_IF

CASE A5_sequence OF
	// INITIATE --------------------------------------------------------------------------------------------------------------		
	0:
		process_A := 0;
		process_B := 0;
		process_C := 0;
		process_D := 0;
		process_E := 0;
		process_F := 0;
		process_G := 0;
		process_H := 0;
		process_I := 0;
		process_J := 0;
		process_K := 0;
		
		JigTimerA (IN:= FALSE);
		JigTimerB (IN:= FALSE);
		JigTimerC (IN:= FALSE);
		TTTimer	  (IN:= FALSE);
		
		AUTO_MODE.JIGA_ErrorState 	:= FALSE;
		AUTO_MODE.JIGB_ErrorState 	:= FALSE;
		AUTO_MODE.JIGC_ErrorState 	:= FALSE;
		AUTO_MODE.TT_ErrorState 	:= FALSE;
		
		AUTO_MODE.processnameA5 := CONCAT(MSG.COMP_A5,MSG.ACTION_INIT);
		LOGPROCESS( spLogComp	 := MSG.COMP_A5, 
		 			spLogAction	 := MSG.ACTION_INIT, 
		 			spLogStatus	 := MSG.STATUS_DONE,
	 	 		 	plogFlag	 := TRUE);
	
		A5_sequence := 1;
		
	// IF RACK PICK (KR5) --------------------------------------------------------------------------------------------------------------		
	1:
		IF process_A = 0 THEN
			Bit1 := 3; 
			Bit2 := 5; //205
			IF 	KR3.Idle AND 
				KR5.Idle AND 
				GVL.JIGA_Standby AND
				NOT AUTO_MODE.JIGA_LOAD AND
				NOT AUTO_MODE.IF_PICK THEN
						KR5.bOutBit[ Bit1,Bit2 ] := TRUE;
						AUTO_MODE.IF_PICK := TRUE;
						process_A := 1;
						AUTO_MODE.processnameA5 := CONCAT(MSG.COMP_A5,MSG.ACTION_IF_A5);
						AUTO_MODE.processnameA5 := CONCAT(AUTO_MODE.processnameA5,MSG.STATUS_RUN);
						LOGPROCESS( spLogComp	 := MSG.COMP_A5, 
									spLogAction	 := MSG.ACTION_IF_A5, 
									spLogStatus	 := MSG.STATUS_RUN,
									plogFlag	 := TRUE);
						RETURN;
			END_IF
		ELSIF process_A = 1 THEN
			KR5.bOutBit[ Bit1,Bit2 ] := TRUE; 
			IF KR5.bInBit[ Bit1,Bit2 ] THEN
				KR5.bOutBit[ Bit1,Bit2 ] := FALSE; 
				process_A := 2;
				AUTO_MODE.processnameA5 := CONCAT(MSG.COMP_A5,MSG.ACTION_IF_A5);
				AUTO_MODE.processnameA5 := CONCAT(AUTO_MODE.processnameA5,MSG.STATUS_ACK);
				LOGPROCESS( spLogComp	 := MSG.COMP_A5, 
							spLogAction	 := MSG.ACTION_IF_A5, 
							spLogStatus	 := MSG.STATUS_ACK,
							plogFlag	 := TRUE);
				RETURN;
			END_IF	
		ELSIF process_A = 2 THEN
			KR5.bOutBit[ Bit1,Bit2 ] := FALSE; 
			IF NOT KR5.bInBit[ Bit1,Bit2 ] THEN
				process_A:= 3;
				AUTO_MODE.processnameA5 := CONCAT(MSG.COMP_A5,MSG.ACTION_IF_A5);
				AUTO_MODE.processnameA5 := CONCAT(AUTO_MODE.processnameA5,MSG.STATUS_DONE);
				LOGPROCESS( spLogComp	 := MSG.COMP_A5, 
							spLogAction	 := MSG.ACTION_IF_A5, 
							spLogStatus	 := MSG.STATUS_DONE,
							plogFlag	 := TRUE);
				RETURN;
			END_IF	
		ELSIF process_A = 3 THEN
			IF KR5.Idle THEN
				process_A := 4;
				A5_sequence := 2;
				AUTO_MODE.next_step := FALSE;
				AUTO_MODE.processnameA5 := CONCAT(MSG.COMP_A5,MSG.ACTION_IF_A5);
				AUTO_MODE.processnameA5 := CONCAT(AUTO_MODE.processnameA5,MSG.STATUS_COMP);
				LOGPROCESS( spLogComp	 := MSG.COMP_A5, 
							spLogAction	 := MSG.ACTION_IF_A5, 
							spLogStatus	 := MSG.STATUS_COMP,
							plogFlag	 := TRUE);
			END_IF
		END_IF	
		
	// PLACE TO JIG A (KR5) --------------------------------------------------------------------------------------------------------------		
	2:
		IF process_J = 0 THEN
			Bit1 := 3; 
			Bit2 := 0; //200
			IF 	KR3.Idle AND 
				KR5.Idle AND
				GVL.JIGA_Standby AND 
				AUTO_MODE.IF_PICK AND 
				NOT AUTO_MODE.JIGA_LOAD THEN 
						KR5.bOutBit[ Bit1,Bit2 ] := TRUE;
						AUTO_MODE.JIGA_LOAD := TRUE;
						process_J := 1;
						AUTO_MODE.processnameA5 := CONCAT(MSG.COMP_A5,MSG.ACTION_JIGA_PLACE);
						AUTO_MODE.processnameA5 := CONCAT(AUTO_MODE.processnameA5,MSG.STATUS_RUN);
						LOGPROCESS( spLogComp	 := MSG.COMP_A5, 
									spLogAction	 := MSG.ACTION_JIGA_PLACE, 
									spLogStatus	 := MSG.STATUS_RUN,
									plogFlag	 := TRUE);
						RETURN;
			END_IF
		ELSIF process_J = 1 THEN
			KR5.bOutBit[ Bit1,Bit2 ] := TRUE;
			IF NOT KR5.bInBit[ Bit1,Bit2 ] THEN
				KR5.bOutBit[ Bit1,Bit2 ] := FALSE;
				process_J := 2;
				AUTO_MODE.processnameA5 := CONCAT(MSG.COMP_A5,MSG.ACTION_JIGA_PLACE);
				AUTO_MODE.processnameA5 := CONCAT(AUTO_MODE.processnameA5,MSG.STATUS_ACK);
				LOGPROCESS( spLogComp	 := MSG.COMP_A5, 
							spLogAction	 := MSG.ACTION_JIGA_PLACE, 
							spLogStatus	 := MSG.STATUS_ACK,
							plogFlag	 := TRUE);
				RETURN;
			END_IF	
		ELSIF process_J = 2 THEN
			KR5.bOutBit[ Bit1,Bit2 ] := FALSE;
			IF KR5.bInBit[ Bit1,Bit2 ] THEN
				process_J:= 3;
				AUTO_MODE.processnameA5 := CONCAT(MSG.COMP_A5,MSG.ACTION_JIGA_PLACE);
				AUTO_MODE.processnameA5 := CONCAT(AUTO_MODE.processnameA5,MSG.STATUS_DONE);
				LOGPROCESS( spLogComp	 := MSG.COMP_A5, 
							spLogAction	 := MSG.ACTION_JIGA_PLACE, 
							spLogStatus	 := MSG.STATUS_DONE,
							plogFlag	 := TRUE);
				RETURN;
			END_IF	
		ELSIF process_J = 3 THEN
			IF 	KR5.Idle AND  
				AUTO_MODE.JIGA_LOAD AND
				NOT GVL.JIGA_Standby THEN
						AUTO_MODE.IF_PICK := FALSE;
						process_J := 4;
						A5_sequence := 3;
						AUTO_MODE.next_step := FALSE;
						AUTO_MODE.processnameA5 := CONCAT(MSG.COMP_A5,MSG.ACTION_JIGA_PLACE);
						AUTO_MODE.processnameA5 := CONCAT(AUTO_MODE.processnameA5,MSG.STATUS_COMP);
						LOGPROCESS( spLogComp	 := MSG.COMP_A5, 
									spLogAction	 := MSG.ACTION_JIGA_PLACE, 
									spLogStatus	 := MSG.STATUS_COMP,
									plogFlag	 := TRUE);
			END_IF
		END_IF	
	
	// JIG A CLAMP -----------------------------------------------------------------------------------------------------------------------
	3:
		IF NOT AUTO_MODE.Halt_Production THEN
			GVL.JIGA_Clamp := TRUE;
			GVL.JIGA_Release := FALSE;
			JigTimerA(IN := TRUE, PT := JIG_ErrorTime);
		END_IF
		//insert Jig safety check here 
		
		IF JigTimerA.Q THEN
			AUTO_MODE.JIGA_ErrorState := TRUE;
			IF GVL.ClearError THEN
				JigTimerA(IN:= FALSE);
				GVL.ClearError := FALSE;
			ELSE
				AUTO_MODE.Halt_Production := TRUE;
				AUTO_MODE.processnameA5 := CONCAT(MSG.COMP_A5,MSG.ACTION_JIGA_CLAMP);
				AUTO_MODE.processnameA5 := CONCAT(AUTO_MODE.processnameA5,MSG.STATUS_ERROR);
				LOGPROCESS( spLogComp	 := MSG.COMP_A5, 
							spLogAction	 := MSG.ACTION_JIGA_CLAMP, 
							spLogStatus	 := MSG.STATUS_ERROR,
							plogFlag	 := TRUE);
			END_IF
		ELSIF GVL.JIGA_Ready THEN
			JigTimerA(IN := FALSE);
			AUTO_MODE.JIGA_ErrorState := FALSE;
			AUTO_MODE.next_step := FALSE;
			AUTO_MODE.processnameA5 := CONCAT(MSG.COMP_A5,MSG.ACTION_JIGA_CLAMP);
			AUTO_MODE.processnameA5 := CONCAT(AUTO_MODE.processnameA5,MSG.STATUS_DONE);
			LOGPROCESS( spLogComp	 := MSG.COMP_A5, 
						spLogAction	 := MSG.ACTION_JIGA_CLAMP, 
						spLogStatus	 := MSG.STATUS_COMP,
						plogFlag	 := TRUE);
			IF GVL.KR2_bypass THEN
				process_B	:= 3;	
				A5_sequence := 4;
			ELSE	
				process_B	:= 0;	
				A5_sequence := 4;
			END_IF
		END_IF
		
	// JIG A WELDING(KR3) ------------------------------------------------------------------------------------------------------------------
	4:
		IF process_B = 0 THEN
			Bit1 := 3; 
			Bit2 := 0; //300
			IF 	KR3.Idle AND 
//				KR5.Idle AND
				GVL.JIGA_Ready AND  
				NOT AUTO_MODE.JIGA_WELDING AND 
				NOT AUTO_MODE.JIGB_WELDING THEN
						KR3.bOutBit[ Bit1,Bit2 ] := TRUE;
						AUTO_MODE.JIGA_WELDING := TRUE;
						process_B := 1;
						AUTO_MODE.processnameA5 := CONCAT(MSG.COMP_A5,MSG.ACTION_JIGA_WELDING);
						AUTO_MODE.processnameA5 := CONCAT(AUTO_MODE.processnameA5,MSG.STATUS_RUN);
						LOGPROCESS( spLogComp	 := MSG.COMP_A5, 
									spLogAction	 := MSG.ACTION_JIGA_WELDING, 
									spLogStatus	 := MSG.STATUS_RUN,
									plogFlag	 := TRUE);
									RETURN;
			END_IF
		ELSIF process_B = 1 THEN 
			KR3.bOutBit[ Bit1,Bit2 ] := TRUE;
			IF NOT KR3.bInBit[ Bit1,Bit2 ] THEN
				KR3.bOutBit[ Bit1,Bit2 ] := FALSE;	
				process_B := 2;
				AUTO_MODE.processnameA5 := CONCAT(MSG.COMP_A5,MSG.ACTION_JIGA_WELDING);
				AUTO_MODE.processnameA5 := CONCAT(AUTO_MODE.processnameA5,MSG.STATUS_ACK);
				LOGPROCESS( spLogComp	 := MSG.COMP_A5, 
							spLogAction	 := MSG.ACTION_JIGA_WELDING, 
							spLogStatus	 := MSG.STATUS_ACK,
							plogFlag	 := TRUE);
				RETURN;
			END_IF
		ELSIF process_B = 2 THEN 
			KR3.bOutBit[ Bit1,Bit2 ] := FALSE;
			IF KR3.bInBit[ Bit1,Bit2 ] THEN
				process_B := 3;
				AUTO_MODE.processnameA5 := CONCAT(MSG.COMP_A5,MSG.ACTION_JIGA_WELDING);
				AUTO_MODE.processnameA5 := CONCAT(AUTO_MODE.processnameA5,MSG.STATUS_DONE);
				LOGPROCESS( spLogComp	 := MSG.COMP_A5, 
							spLogAction	 := MSG.ACTION_JIGA_WELDING, 
							spLogStatus	 := MSG.STATUS_DONE,
							plogFlag	 := TRUE);
				RETURN;
			END_IF
		ELSIF process_B = 3 THEN
			IF KR3.Idle THEN
				AUTO_MODE.JIGA_WELDING := FALSE;
				GVL.JIGA_Clamp := FALSE;
				GVL.JIGA_Release := TRUE;
				JigTimerA(IN := FALSE);
				AUTO_MODE.processnameA5 := CONCAT(MSG.COMP_A5,MSG.ACTION_JIGA_RELEASE);
				AUTO_MODE.processnameA5 := CONCAT(AUTO_MODE.processnameA5,MSG.STATUS_DONE);
				LOGPROCESS( spLogComp	 := MSG.COMP_A5, 
							spLogAction	 := MSG.ACTION_JIGA_RELEASE, 
							spLogStatus	 := MSG.STATUS_DONE,
							plogFlag	 := TRUE);
				process_B := 4;
				AUTO_MODE.processnameA5 := CONCAT(MSG.COMP_A5,MSG.ACTION_JIGA_WELDING);
				AUTO_MODE.processnameA5 := CONCAT(AUTO_MODE.processnameA5,MSG.STATUS_COMP);
				LOGPROCESS( spLogComp	 := MSG.COMP_A5, 
							spLogAction	 := MSG.ACTION_JIGA_WELDING, 
							spLogStatus	 := MSG.STATUS_COMP,
							plogFlag	 := TRUE);
			END_IF
		ELSIF process_B = 4 THEN
			IF NOT AUTO_MODE.Halt_Production THEN
				GVL.JIGA_Clamp 		:= FALSE;
				GVL.JIGA_Release 	:= TRUE;
				JigTimerA(IN := TRUE, PT := JIG_ErrorTime);
			END_IF
			//insert Jig safety check here ------------------------------
			IF JigTimerA.Q THEN
				AUTO_MODE.JIGA_ErrorState := TRUE;
				IF GVL.ClearError THEN
					JigTimerA(IN:= FALSE);
					GVL.ClearError := FALSE;
				ELSE
					AUTO_MODE.Halt_Production := TRUE;
					AUTO_MODE.processnameA5 := CONCAT(MSG.COMP_A5,MSG.ACTION_JIGA_RELEASE);
					AUTO_MODE.processnameA5 := CONCAT(AUTO_MODE.processnameA5,MSG.STATUS_ERROR);
					LOGPROCESS( spLogComp	 := MSG.COMP_A5, 
								spLogAction	 := MSG.ACTION_JIGA_RELEASE, 
								spLogStatus	 := MSG.STATUS_ERROR,
								plogFlag	 := TRUE);
				END_IF
			ELSIF GVL.JIGA_Complete THEN
				JigTimerA(IN:= FALSE);
				AUTO_MODE.JIGA_ErrorState := FALSE;
				process_B := 5;
				A5_sequence := 5;
				AUTO_MODE.next_step := FALSE;
				AUTO_MODE.processnameA5 := CONCAT(MSG.COMP_A5,MSG.ACTION_JIGA_COMPLETE);
				AUTO_MODE.processnameA5 := CONCAT(AUTO_MODE.processnameA5,MSG.STATUS_COMP);
				LOGPROCESS( spLogComp	 := MSG.COMP_A5, 
							spLogAction	 := MSG.ACTION_JIGA_COMPLETE, 
							spLogStatus	 := MSG.STATUS_COMP,
							plogFlag	 := TRUE);
			END_IF
		END_IF
		
	// JIG A TO JIG B {KR5} -----------------------------------------------------------------------------------------------------------------
	5: 
		IF process_C = 0 THEN
			Bit1 := 3;
			Bit2 := 1; //201
			IF 	KR3.Idle AND 
				KR5.Idle AND 
				GVL.JIGB_Standby AND 
				NOT GVL.JIGA_Ready AND 
				NOT AUTO_MODE.JIGB_LOAD AND 
				NOT AUTO_MODE.JIGA_WELDING AND 
				NOT AUTO_MODE.JIGB_WELDING AND 
				NOT AUTO_MODE.JIGC_WELDING THEN
						AUTO_MODE.JIGB_LOAD := TRUE;
						KR5.bOutBit[ Bit1, Bit2 ] := TRUE;
						process_C := 1;
						AUTO_MODE.processnameA5 := CONCAT(MSG.COMP_A5,MSG.ACTION_JIGA_TO_JIGB);
						AUTO_MODE.processnameA5 := CONCAT(AUTO_MODE.processnameA5,MSG.STATUS_RUN);
						LOGPROCESS( spLogComp	 := MSG.COMP_A5, 
									spLogAction	 := MSG.ACTION_JIGA_TO_JIGB, 
									spLogStatus	 := MSG.STATUS_RUN,
									plogFlag	 := TRUE);
						RETURN;
			END_IF
		ELSIF process_C = 1 THEN 
			KR5.bOutBit [ Bit1, Bit2 ] := TRUE;
			IF KR5.bInBit[ Bit1, Bit2 ] THEN
				KR5.bOutBit[ Bit1, Bit2 ] := FALSE;
				process_C := 2;
				AUTO_MODE.processnameA5 := CONCAT(MSG.COMP_A5,MSG.ACTION_JIGA_TO_JIGB);
				AUTO_MODE.processnameA5 := CONCAT(AUTO_MODE.processnameA5,MSG.STATUS_ACK);
				LOGPROCESS( spLogComp	 := MSG.COMP_A5, 
							spLogAction	 := MSG.ACTION_JIGA_TO_JIGB, 
							spLogStatus	 := MSG.STATUS_ACK,
							plogFlag	 := TRUE);
				RETURN;
			END_IF
		ELSIF process_C = 2 THEN 
			KR5.bOutBit[ Bit1, Bit2 ] := FALSE;
			IF NOT KR5.bInBit[ Bit1, Bit2 ] THEN
				process_C := 3;
				AUTO_MODE.processnameA5 := CONCAT(MSG.COMP_A5,MSG.ACTION_JIGA_TO_JIGB);
				AUTO_MODE.processnameA5 := CONCAT(AUTO_MODE.processnameA5,MSG.STATUS_DONE);
				LOGPROCESS( spLogComp	 := MSG.COMP_A5, 
							spLogAction	 := MSG.ACTION_JIGA_TO_JIGB, 
							spLogStatus	 := MSG.STATUS_DONE,
							plogFlag	 := TRUE);
				RETURN;
			END_IF
		ELSIF process_C = 3 THEN
			IF 	KR5.Idle AND 
				NOT GVL.JIGB_Standby THEN
						AUTO_MODE.JIGA_LOAD := FALSE;
						process_C := 4;
						A5_sequence := 6;
						AUTO_MODE.next_step := FALSE;
						AUTO_MODE.processnameA5 := CONCAT(MSG.COMP_A5,MSG.ACTION_JIGA_TO_JIGB);
						AUTO_MODE.processnameA5 := CONCAT(AUTO_MODE.processnameA5,MSG.STATUS_COMP);
						LOGPROCESS( spLogComp	 := MSG.COMP_A5, 
									spLogAction	 := MSG.ACTION_JIGA_TO_JIGB, 
									spLogStatus	 := MSG.STATUS_COMP,
									plogFlag	 := TRUE);
			END_IF
		END_IF
		
	//	JIG B CLAMP	-----------------------------------------------------------------------------------------------------------------------
	6:
		IF NOT AUTO_MODE.Halt_Production THEN
			GVL.JIGB_Clamp := TRUE;
			GVL.JIGB_Release := FALSE;
			JigTimerB(IN := TRUE, PT := JIG_ErrorTime);
		END_IF
		//insert Jig safety check here ------------------------------
		IF JigTimerB.Q THEN
			AUTO_MODE.JIGB_ErrorState := TRUE;
			IF GVL.ClearError THEN
				JigTimerB(IN:= FALSE);
				GVL.ClearError := FALSE;
			ELSE
				AUTO_MODE.Halt_Production := TRUE;
			AUTO_MODE.processnameA5 := CONCAT(MSG.COMP_A5,MSG.ACTION_JIGB_CLAMP);
			AUTO_MODE.processnameA5 := CONCAT(AUTO_MODE.processnameA5,MSG.STATUS_ERROR);
			LOGPROCESS( spLogComp	 := MSG.COMP_A5, 
						spLogAction	 := MSG.ACTION_JIGB_CLAMP, 
						spLogStatus	 := MSG.STATUS_DONE,
						plogFlag	 := TRUE);
			END_IF
		ELSIF GVL.JIGB_Ready THEN
			JigTimerB(IN:= FALSE);
			AUTO_MODE.JIGB_ErrorState := FALSE;
			AUTO_MODE.next_step := FALSE;
			AUTO_MODE.processnameA5 := CONCAT(MSG.COMP_A5,MSG.ACTION_JIGB_CLAMP);
			AUTO_MODE.processnameA5 := CONCAT(AUTO_MODE.processnameA5,MSG.STATUS_DONE);
			LOGPROCESS( spLogComp	 := MSG.COMP_A5, 
						spLogAction	 := MSG.ACTION_JIGB_CLAMP, 
						spLogStatus	 := MSG.STATUS_DONE,
						plogFlag	 := TRUE);
			IF GVL.KR2_bypass THEN
				process_D	:= 3;	
				A5_sequence := 7;
			ELSE	
				process_D	:= 0;	
				A5_sequence := 7;
			END_IF
		END_IF
		
	// JIG B WELDING (KR3) -------------------------------------------------------------------------------------------------------------	
	7:
		IF process_D = 0 THEN
			Bit1 := 3;
			Bit2 := 1; //301
			IF 	KR3.Idle AND 
				GVL.JIGB_Ready AND
				NOT AUTO_MODE.JIGA_WELDING AND 
				NOT AUTO_MODE.JIGB_WELDING THEN
						KR3.bOutBit[ Bit1, Bit2 ] := TRUE;
						AUTO_MODE.JIGB_WELDING := TRUE;
						process_D := 1;
						AUTO_MODE.processnameA5 := CONCAT(MSG.COMP_A5,MSG.ACTION_JIGB_WELDING);
						AUTO_MODE.processnameA5 := CONCAT(AUTO_MODE.processnameA5,MSG.STATUS_RUN);
						LOGPROCESS( spLogComp	 := MSG.COMP_A5, 
									spLogAction	 := MSG.ACTION_JIGB_WELDING, 
									spLogStatus	 := MSG.STATUS_RUN,
									plogFlag	 := TRUE);
				RETURN;
			END_IF
		ELSIF process_D = 1 THEN
			KR3.bOutBit[ Bit1, Bit2 ] := TRUE;
			IF KR3.bInBit[ Bit1, Bit2 ] THEN
				KR3.bOutBit[ Bit1, Bit2 ] := FALSE;
				process_D := 2;
				AUTO_MODE.processnameA5 := CONCAT(MSG.COMP_A5,MSG.ACTION_JIGB_WELDING);
				AUTO_MODE.processnameA5 := CONCAT(AUTO_MODE.processnameA5,MSG.STATUS_ACK);
				LOGPROCESS( spLogComp	 := MSG.COMP_A5, 
							spLogAction	 := MSG.ACTION_JIGB_WELDING, 
							spLogStatus	 := MSG.STATUS_ACK,
							plogFlag	 := TRUE);
				RETURN;
			END_IF
		ELSIF process_D = 2 THEN
			KR3.bOutBit[ Bit1, Bit2 ] := FALSE;
			IF NOT KR3.bInBit[ Bit1, Bit2 ] THEN
				process_D := 3;
				AUTO_MODE.Run_Next_Rack := TRUE;
				AUTO_MODE.processnameA5 := CONCAT(MSG.COMP_A5,MSG.ACTION_JIGB_WELDING);
				AUTO_MODE.processnameA5 := CONCAT(AUTO_MODE.processnameA5,MSG.STATUS_DONE);
				LOGPROCESS( spLogComp	 := MSG.COMP_A5, 
							spLogAction	 := MSG.ACTION_JIGB_WELDING, 
							spLogStatus	 := MSG.STATUS_DONE,
							plogFlag	 := TRUE);
				RETURN;
			END_IF
		ELSIF process_D = 3 THEN
			IF KR3.Idle THEN
				AUTO_MODE.JIGB_WELDING := FALSE;
				GVL.JIGB_Clamp := FALSE;
				GVL.JIGB_Release := TRUE;
				JigTimerB(IN:= FALSE);
				AUTO_MODE.processnameA5 := CONCAT(MSG.COMP_A5,MSG.ACTION_JIGB_RELEASE);
				AUTO_MODE.processnameA5 := CONCAT(AUTO_MODE.processnameA5,MSG.STATUS_DONE);
				LOGPROCESS( spLogComp	 := MSG.COMP_A5, 
							spLogAction	 := MSG.ACTION_JIGB_RELEASE, 
							spLogStatus	 := MSG.STATUS_DONE,
							plogFlag	 := TRUE);
				process_D := 4;
				AUTO_MODE.processnameA5 := CONCAT(MSG.COMP_A5,MSG.ACTION_JIGB_WELDING);
				AUTO_MODE.processnameA5 := CONCAT(AUTO_MODE.processnameA5,MSG.STATUS_COMP);
				LOGPROCESS( spLogComp	 := MSG.COMP_A5, 
							spLogAction	 := MSG.ACTION_JIGB_WELDING, 
							spLogStatus	 := MSG.STATUS_COMP,
							plogFlag	 := TRUE);
			END_IF
		ELSIF process_D = 4 THEN
			IF NOT AUTO_MODE.Halt_Production THEN
				GVL.JIGB_Clamp 		:= FALSE;
				GVL.JIGB_Release 	:= TRUE;
				JigTimerB(IN := TRUE, PT := JIG_ErrorTime);
			END_IF
			//insert Jig safety check here ------------------------------
			IF JigTimerB.Q THEN
				AUTO_MODE.JIGB_ErrorState := TRUE;
				IF GVL.ClearError THEN
					JigTimerB(IN:= FALSE);
					GVL.ClearError := FALSE;
				ELSE
					AUTO_MODE.Halt_Production := TRUE;
					AUTO_MODE.processnameA5 := CONCAT(MSG.COMP_A5,MSG.ACTION_JIGB_RELEASE);
					AUTO_MODE.processnameA5 := CONCAT(AUTO_MODE.processnameA5,MSG.STATUS_ERROR);
					LOGPROCESS( spLogComp	 := MSG.COMP_A5, 
								spLogAction	 := MSG.ACTION_JIGB_RELEASE, 
								spLogStatus	 := MSG.STATUS_ERROR,
								plogFlag	 := TRUE);
				END_IF
			ELSIF GVL.JIGB_Complete THEN
				JigTimerB(IN:= FALSE);
				AUTO_MODE.JIGB_ErrorState := FALSE;
				process_D := 5;
				A5_sequence := 8;
				AUTO_MODE.next_step := FALSE;
				AUTO_MODE.processnameA5 := CONCAT(MSG.COMP_A5,MSG.ACTION_JIGB_COMPLETE);
				AUTO_MODE.processnameA5 := CONCAT(AUTO_MODE.processnameA5,MSG.STATUS_COMP);
				LOGPROCESS( spLogComp	 := MSG.COMP_A5, 
							spLogAction	 := MSG.ACTION_JIGB_COMPLETE, 
							spLogStatus	 := MSG.STATUS_COMP,
							plogFlag	 := TRUE);
			END_IF
		END_IF
		
	// JIG B TO TWINTORCH (KR5) -------------------------------------------------------------------------------------------------------------
	8: 
		IF process_E = 0 THEN
			Bit1 := 3;
			Bit2 := 2; //302
//			IF 	KR3.Idle AND 
			IF	KR5.Idle AND
				GVL.TTorch_Standy AND 
				NOT AUTO_MODE.IF_PICK AND
				NOT AUTO_MODE.IF_PICK AND
				NOT AUTO_MODE.TT_LOAD AND 
				NOT GVL.JIGB_Ready AND
				NOT AUTO_MODE.JIGA_WELDING AND 
				NOT AUTO_MODE.JIGB_WELDING AND 
				NOT AUTO_MODE.TT_WELDING THEN
						AUTO_MODE.TT_LOAD := TRUE;
						KR5.bOutBit[ Bit1, Bit2 ] := TRUE;
						process_E := 1;
						AUTO_MODE.processnameA5 := CONCAT(MSG.COMP_A5,MSG.ACTION_JIGB_TO_TT);
						AUTO_MODE.processnameA5 := CONCAT(AUTO_MODE.processnameA5,MSG.STATUS_RUN);
						LOGPROCESS( spLogComp	 := MSG.COMP_A5, 
									spLogAction	 := MSG.ACTION_JIGB_TO_TT, 
									spLogStatus	 := MSG.STATUS_RUN,
									plogFlag	 := TRUE);
						RETURN;
			END_IF
		ELSIF process_E = 1 THEN
			KR5.bOutBit[ Bit1, Bit2 ] := TRUE;
			IF KR5.bInBit[ Bit1, Bit2 ] THEN
				KR5.bOutBit[ Bit1, Bit2 ] := FALSE;
				process_E := 2;
				AUTO_MODE.processnameA5 := CONCAT(MSG.COMP_A5,MSG.ACTION_JIGB_TO_TT);
				AUTO_MODE.processnameA5 := CONCAT(AUTO_MODE.processnameA5,MSG.STATUS_ACK);
				LOGPROCESS( spLogComp	 := MSG.COMP_A5, 
							spLogAction	 := MSG.ACTION_JIGB_TO_TT, 
							spLogStatus	 := MSG.STATUS_ACK,
							plogFlag	 := TRUE);
				RETURN;
			END_IF
		ELSIF process_E = 2 THEN
			KR5.bOutBit[ Bit1, Bit2 ] := FALSE;
			IF NOT KR5.bInBit[ Bit1, Bit2 ] THEN
				process_E := 3;
				AUTO_MODE.processnameA5 := CONCAT(MSG.COMP_A5,MSG.ACTION_JIGB_TO_TT);
				AUTO_MODE.processnameA5 := CONCAT(AUTO_MODE.processnameA5,MSG.STATUS_DONE);
				LOGPROCESS( spLogComp	 := MSG.COMP_A5, 
							spLogAction	 := MSG.ACTION_JIGB_TO_TT, 
							spLogStatus	 := MSG.STATUS_DONE,
							plogFlag	 := TRUE);
				RETURN;
			END_IF
		ELSIF process_E = 3 THEN
			IF KR5.Idle THEN
				AUTO_MODE.JIGB_LOAD := FALSE;
				process_E := 4;
				A5_sequence := 9;
				AUTO_MODE.next_step := FALSE;
//				AUTO_MODE.Run_Next_Rack :=TRUE;
				AUTO_MODE.processnameA5 := CONCAT(MSG.COMP_A5,MSG.ACTION_JIGB_TO_TT);
				AUTO_MODE.processnameA5 := CONCAT(AUTO_MODE.processnameA5,MSG.STATUS_COMP);
				LOGPROCESS( spLogComp	 := MSG.COMP_A5, 
							spLogAction	 := MSG.ACTION_JIGB_TO_TT, 
							spLogStatus	 := MSG.STATUS_COMP,
							plogFlag	 := TRUE);
			END_IF
		END_IF	
	
	// TWINTORCH WELDING -------------------------------------------------------------------------------------------------------------	
	9:
		//insert Jig safety check here ------------------------------
		IF NOT GVL.TTorch_Standy THEN
			GVL.TTorch_Run := TRUE;
			AUTO_MODE.TT_WELDING := TRUE;
			A5_sequence := 10;
			TTTimer(IN := TRUE, PT := TT_ErrorTime);
			AUTO_MODE.processnameA5 := CONCAT(MSG.COMP_A5,MSG.ACTION_TT_RUN);
			AUTO_MODE.processnameA5 := CONCAT(AUTO_MODE.processnameA5,MSG.STATUS_RUN);
			LOGPROCESS( spLogComp	 := MSG.COMP_A5, 
						spLogAction	 := MSG.ACTION_TT_RUN, 
						spLogStatus	 := MSG.STATUS_RUN,
						plogFlag	 := TRUE);
			RETURN;
		END_IF
	// TWINTORCH WELD COMPLETE -------------------------------------------------------------------------------------------------------------		
	10:
		
		//insert Jig safety check here ------------------------------
		IF TTTimer.Q THEN
			AUTO_MODE.TT_ErrorState := TRUE;
			IF GVL.ClearError THEN
				TTTimer(IN:= FALSE);
				GVL.ClearError := FALSE;
			ELSE
				AUTO_MODE.Halt_Production := TRUE;
				AUTO_MODE.processnameA5 := CONCAT(MSG.COMP_A5,MSG.ACTION_TT_RUN);
				AUTO_MODE.processnameA5 := CONCAT(AUTO_MODE.processnameA5,MSG.STATUS_ERROR);
				LOGPROCESS( spLogComp	 := MSG.COMP_A5, 
							spLogAction	 := MSG.ACTION_TT_RUN, 
							spLogStatus	 := MSG.STATUS_ERROR,
							plogFlag	 := TRUE);
			END_IF
		ELSIF GVL.TTorch_Complete THEN
			TTTimer(IN:= FALSE);
			AUTO_MODE.TT_ErrorState := FALSE;
			GVL.TTorch_Run := FALSE;
			AUTO_MODE.TT_WELDING := FALSE;
			A5_sequence := 11;
			AUTO_MODE.next_step := FALSE;
			AUTO_MODE.processnameA5 := CONCAT(MSG.COMP_A5,MSG.ACTION_TT_RUN);
			AUTO_MODE.processnameA5 := CONCAT(AUTO_MODE.processnameA5,MSG.STATUS_DONE);
			LOGPROCESS( spLogComp	 := MSG.COMP_A5, 
						spLogAction	 := MSG.ACTION_TT_RUN, 
						spLogStatus	 := MSG.STATUS_DONE,
						plogFlag	 := TRUE);
			RETURN;
		END_IF
		
	// TWINTORCH TO JIG C (KR5)	-------------------------------------------------------------------------------------------------------
	11:
		IF process_F = 0 THEN
			Bit1 := 3;
			Bit2 := 3; //203
			IF 	KR5.Idle AND 
				KR4.Idle AND 
				GVL.JIGC_Standby AND 
				NOT AUTO_MODE.JIGC_LOAD AND
				NOT AUTO_MODE.JIGC_WELDING AND 
				NOT AUTO_MODE.TT_WELDING  THEN
						KR5.bOutBit[ Bit1, Bit2 ] := TRUE;
						process_F := 1;
						AUTO_MODE.processnameA5 := CONCAT(MSG.COMP_A5,MSG.ACTION_TT_TO_JIGC);
						AUTO_MODE.processnameA5 := CONCAT(AUTO_MODE.processnameA5,MSG.STATUS_RUN);
						LOGPROCESS( spLogComp	 := MSG.COMP_A5, 
									spLogAction	 := MSG.ACTION_TT_TO_JIGC, 
									spLogStatus	 := MSG.STATUS_RUN,
									plogFlag	 := TRUE);
						RETURN;
			END_IF
		ELSIF process_F = 1 THEN
			KR5.bOutBit[ Bit1, Bit2 ] := TRUE;
			IF KR5.bInBit[ Bit1, Bit2 ] THEN
				KR5.bOutBit[ Bit1, Bit2 ] := FALSE;	
				process_F := 2;
				AUTO_MODE.processnameA5 := CONCAT(MSG.COMP_A5,MSG.ACTION_TT_TO_JIGC);
				AUTO_MODE.processnameA5 := CONCAT(AUTO_MODE.processnameA5,MSG.STATUS_ACK);
				LOGPROCESS( spLogComp	 := MSG.COMP_A5, 
							spLogAction	 := MSG.ACTION_TT_TO_JIGC, 
							spLogStatus	 := MSG.STATUS_ACK,
							plogFlag	 := TRUE);
				RETURN;
			END_IF
		ELSIF process_F = 2 THEN
			KR5.bOutBit[ Bit1, Bit2 ] := FALSE;	
			IF NOT KR5.bInBit[ Bit1, Bit2 ] THEN
				process_F := 3;
				AUTO_MODE.processnameA5 := CONCAT(MSG.COMP_A5,MSG.ACTION_TT_TO_JIGC);
				AUTO_MODE.processnameA5 := CONCAT(AUTO_MODE.processnameA5,MSG.STATUS_DONE);
				LOGPROCESS( spLogComp	 := MSG.COMP_A5, 
							spLogAction	 := MSG.ACTION_TT_TO_JIGC, 
							spLogStatus	 := MSG.STATUS_DONE,
							plogFlag	 := TRUE);
				RETURN;
			END_IF
		ELSIF process_F = 3 THEN
			IF KR5.Idle AND NOT GVL.JIGC_Standby THEN
				AUTO_MODE.JIGC_LOAD := TRUE;
				AUTO_MODE.TT_LOAD := FALSE;
				process_F := 4;
				A5_sequence := 12;
				AUTO_MODE.next_step := FALSE;
				AUTO_MODE.processnameA5 := CONCAT(MSG.COMP_A5,MSG.ACTION_TT_TO_JIGC);
				AUTO_MODE.processnameA5 := CONCAT(AUTO_MODE.processnameA5,MSG.STATUS_COMP);
				LOGPROCESS( spLogComp	 := MSG.COMP_A5, 
							spLogAction	 := MSG.ACTION_TT_TO_JIGC, 
							spLogStatus	 := MSG.STATUS_COMP,
							plogFlag	 := TRUE);
			END_IF
		END_IF
	
	// BRACKET TO JIG C (KR2) -------------------------------------------------------------------------------------------------------------
	12:
		Bit1 := 3;
		Bit2 := 0; //200
		IF process_G = 0 THEN
			IF 	KR2.Idle AND 
				KR4.Idle AND 
				GVL.VibBowl_Ready AND
				AUTO_MODE.JIGC_LOAD AND 
				NOT GVL.JIGC_Standby AND 
				NOT AUTO_MODE.CR_PICK AND
				NOT AUTO_MODE.JIGC_PICK AND
				NOT AUTO_MODE.JIGC_WELDING THEN
						KR2.bOutBit[ Bit1, Bit2 ] := TRUE;
						AUTO_MODE.VB_PICK := TRUE;
						process_G := 1;
						AUTO_MODE.processnameA5 := CONCAT(MSG.COMP_A5,MSG.ACTION_VB_TO_JIGC);
						AUTO_MODE.processnameA5 := CONCAT(AUTO_MODE.processnameA5,MSG.STATUS_RUN);
						LOGPROCESS( spLogComp	 := MSG.COMP_A5, 
									spLogAction	 := MSG.ACTION_VB_TO_JIGC, 
									spLogStatus	 := MSG.STATUS_RUN,
									plogFlag	 := TRUE);
						RETURN;
			END_IF
		ELSIF process_G = 1 THEN
			KR2.bOutBit[ Bit1, Bit2 ] := TRUE;
			IF NOT KR2.bInBit[ Bit1, Bit2 ] THEN
				KR2.bOutBit[ Bit1, Bit2 ] := FALSE;
				process_G := 2;
				AUTO_MODE.processnameA5 := CONCAT(MSG.COMP_A5,MSG.ACTION_VB_TO_JIGC);
				AUTO_MODE.processnameA5 := CONCAT(AUTO_MODE.processnameA5,MSG.STATUS_ACK);
				LOGPROCESS( spLogComp	 := MSG.COMP_A5, 
							spLogAction	 := MSG.ACTION_VB_TO_JIGC, 
							spLogStatus	 := MSG.STATUS_ACK,
							plogFlag	 := TRUE);
				RETURN;
			END_IF
		ELSIF process_G = 2 THEN
			KR2.bOutBit[ Bit1, Bit2 ] := FALSE;
			IF KR2.bInBit[ Bit1, Bit2 ] THEN
				process_G := 3;
				AUTO_MODE.processnameA5 := CONCAT(MSG.COMP_A5,MSG.ACTION_VB_TO_JIGC);
				AUTO_MODE.processnameA5 := CONCAT(AUTO_MODE.processnameA5,MSG.STATUS_DONE);
				LOGPROCESS( spLogComp	 := MSG.COMP_A5, 
							spLogAction	 := MSG.ACTION_VB_TO_JIGC, 
							spLogStatus	 := MSG.STATUS_DONE,
							plogFlag	 := TRUE);
				RETURN;
			END_IF
		ELSIF process_G = 3 THEN 
			IF 	KR2.Idle AND 
				NOT GVL.JIGC_Standby AND 
				AUTO_MODE.JIGC_LOAD THEN
						AUTO_MODE.VB_PICK := FALSE;
						process_G := 4;
						A5_sequence := 13;
						AUTO_MODE.next_step := FALSE;
						AUTO_MODE.processnameA5 := CONCAT(MSG.COMP_A5,MSG.ACTION_VB_TO_JIGC);
						AUTO_MODE.processnameA5 := CONCAT(AUTO_MODE.processnameA5,MSG.STATUS_COMP);
						LOGPROCESS( spLogComp	 := MSG.COMP_A5, 
									spLogAction	 := MSG.ACTION_VB_TO_JIGC, 
									spLogStatus	 := MSG.STATUS_COMP,
									plogFlag	 := TRUE);
			END_IF
		END_IF
		
	// JIG C CLAMP ---------------------------------------------------------------------------------------------------------------
	13:
		IF NOT AUTO_MODE.Halt_Production THEN
			GVL.JIGC_Clamp := TRUE;
			GVL.JIGC_Release := FALSE;
			JigTimerC(IN := TRUE, PT := JIG_ErrorTime);
		END_IF
		//insert Jig safety check here ------------------------------
		IF JigTimerC.Q THEN
			AUTO_MODE.JIGC_ErrorState := TRUE;
			IF GVL.ClearError THEN
				JigTimerC(IN:= FALSE);
				GVL.ClearError := FALSE;
			ELSE
				AUTO_MODE.Halt_Production := TRUE;
				AUTO_MODE.processnameA5 := CONCAT(MSG.COMP_A5,MSG.ACTION_JIGC_CLAMP);
				AUTO_MODE.processnameA5 := CONCAT(AUTO_MODE.processnameA5,MSG.STATUS_ERROR);
				LOGPROCESS( spLogComp	 := MSG.COMP_A5, 
							spLogAction	 := MSG.ACTION_JIGC_CLAMP, 
							spLogStatus	 := MSG.STATUS_ERROR,
							plogFlag	 := TRUE);
			END_IF
		ELSIF GVL.JIGC_Ready THEN
			JigTimerC(IN:= FALSE);
			AUTO_MODE.JIGC_ErrorState := FALSE;
			AUTO_MODE.next_step := FALSE;
			AUTO_MODE.processnameA5 := CONCAT(MSG.COMP_A5,MSG.ACTION_JIGC_CLAMP);
			AUTO_MODE.processnameA5 := CONCAT(AUTO_MODE.processnameA5,MSG.STATUS_DONE);
			LOGPROCESS( spLogComp	 := MSG.COMP_A5, 
						spLogAction	 := MSG.ACTION_JIGC_CLAMP, 
						spLogStatus	 := MSG.STATUS_DONE,
						plogFlag	 := TRUE);
			IF GVL.KR4_bypass THEN
				process_H	:= 3;	
				A5_sequence := 14;
			ELSE	
				process_H	:= 0;	
				A5_sequence := 14;
			END_IF
		END_IF
		
	// JIG C WELDING (KR4) -------------------------------------------------------------------------------------------------------
	14:
		IF process_H = 0 THEN
			Bit1 := 3;
			Bit2 := 0; // 300
			IF 	KR4.Idle AND 
				GVL.JIGC_Ready AND 
				AUTO_MODE.JIGC_LOAD AND
				NOT AUTO_MODE.JIGC_WELDING THEN
						KR4.bOutBit[ Bit1,Bit2 ] := TRUE;
						AUTO_MODE.JIGC_WELDING := TRUE;
						process_H := 1;
						AUTO_MODE.processnameA5 := CONCAT(MSG.COMP_A5,MSG.ACTION_JIGC_WELDING);
						AUTO_MODE.processnameA5 := CONCAT(AUTO_MODE.processnameA5,MSG.STATUS_RUN);
						LOGPROCESS( spLogComp	 := MSG.COMP_A5, 
									spLogAction	 := MSG.ACTION_JIGC_WELDING, 
									spLogStatus	 := MSG.STATUS_RUN,
									plogFlag	 := TRUE);
						RETURN;
			END_IF
		ELSIF process_H = 1 THEN
			KR4.bOutBit[ Bit1,Bit2 ] := TRUE;
			IF NOT KR4.bInBit[ Bit1,Bit2 ] THEN
				KR4.bOutBit[ Bit1,Bit2 ] := FALSE;
				process_H := 2;
				AUTO_MODE.processnameA5 := CONCAT(MSG.COMP_A5,MSG.ACTION_JIGC_WELDING);
				AUTO_MODE.processnameA5 := CONCAT(AUTO_MODE.processnameA5,MSG.STATUS_ACK);
				LOGPROCESS( spLogComp	 := MSG.COMP_A5, 
							spLogAction	 := MSG.ACTION_JIGC_WELDING, 
							spLogStatus	 := MSG.STATUS_ACK,
							plogFlag	 := TRUE);
				RETURN;
			END_IF
		ELSIF process_H = 2 THEN
			KR4.bOutBit[ Bit1,Bit2 ] := FALSE;
			IF KR4.bInBit[ Bit1,Bit2 ] THEN
				process_H := 3;
				AUTO_MODE.processnameA5 := CONCAT(MSG.COMP_A5,MSG.ACTION_JIGC_WELDING);
				AUTO_MODE.processnameA5 := CONCAT(AUTO_MODE.processnameA5,MSG.STATUS_DONE);
				LOGPROCESS( spLogComp	 := MSG.COMP_A5, 
							spLogAction	 := MSG.ACTION_JIGC_WELDING, 
							spLogStatus	 := MSG.STATUS_DONE,
							plogFlag	 := TRUE);
				RETURN;
			END_IF
		ELSIF process_H = 3 THEN
			IF KR4.Idle THEN
				AUTO_MODE.JIGC_WELDING := FALSE;
				GVL.JIGC_Release := TRUE;
				GVL.JIGC_Clamp := FALSE;
				JigTimerC(IN:= FALSE);
				process_H := 4;
				AUTO_MODE.processnameA5 := CONCAT(MSG.COMP_A5,MSG.ACTION_JIGC_WELDING);
				AUTO_MODE.processnameA5 := CONCAT(AUTO_MODE.processnameA5,MSG.STATUS_COMP);
				LOGPROCESS( spLogComp	 := MSG.COMP_A5, 
							spLogAction	 := MSG.ACTION_JIGC_WELDING, 
							spLogStatus	 := MSG.STATUS_COMP,
							plogFlag	 := TRUE);
			END_IF
		ELSIF process_H = 4 THEN
			IF NOT AUTO_MODE.Halt_Production THEN
				GVL.JIGC_Clamp 		:= FALSE;
				GVL.JIGC_Release 	:= TRUE;
				JigTimerC(IN := TRUE, PT := JIG_ErrorTime);
			END_IF
			//insert Jig safety check here ------------------------------
			IF JigTimerC.Q THEN
				AUTO_MODE.JIGC_ErrorState := TRUE;
				IF GVL.ClearError THEN
					JigTimerC(IN:= FALSE);
					GVL.ClearError := FALSE;
				ELSE
					AUTO_MODE.Halt_Production := TRUE;
					AUTO_MODE.processnameA5 := CONCAT(MSG.COMP_A5,MSG.ACTION_JIGC_RELEASE);
					AUTO_MODE.processnameA5 := CONCAT(AUTO_MODE.processnameA5,MSG.STATUS_ERROR);
					LOGPROCESS( spLogComp	 := MSG.COMP_A5, 
								spLogAction	 := MSG.ACTION_JIGC_RELEASE, 
								spLogStatus	 := MSG.STATUS_ERROR,
								plogFlag	 := TRUE);
				END_IF
			ELSIF GVL.JIGC_Complete THEN
				JigTimerC(IN:= FALSE);
				AUTO_MODE.JIGC_ErrorState := FALSE;
				process_H := 5;
				A5_sequence := 15;
				AUTO_MODE.next_step := FALSE;
				AUTO_MODE.processnameA5 := CONCAT(MSG.COMP_A5,MSG.ACTION_JIGC_COMPLETE);
				AUTO_MODE.processnameA5 := CONCAT(AUTO_MODE.processnameA5,MSG.STATUS_COMP);
				LOGPROCESS( spLogComp	 := MSG.COMP_A5, 
							spLogAction	 := MSG.ACTION_JIGC_COMPLETE, 
							spLogStatus	 := MSG.STATUS_COMP,
							plogFlag	 := TRUE);
			END_IF
		END_IF
		
	// JIG C PICK (KR2) -------------------------------------------------------------------------------------------------------
	15: 
		IF process_I = 0 THEN
			Bit1 := 3;
			Bit2 := 2; // 202
			IF 	KR2.Idle AND 
				KR4.Idle AND 
				NOT GVL.JIGC_Ready AND 
				AUTO_MODE.JIGC_LOAD AND 
				NOT AUTO_MODE.JIGC_PICK AND
				NOT AUTO_MODE.CR_PICK THEN
						KR2.bOutBit[ Bit1, Bit2 ] := TRUE;
						AUTO_MODE.JIGC_PICK := TRUE;
						process_I := 1;
						AUTO_MODE.processnameA5 := CONCAT(MSG.COMP_A5,MSG.ACTION_JIGC_PICK);
						AUTO_MODE.processnameA5 := CONCAT(AUTO_MODE.processnameA5,MSG.STATUS_RUN);
						LOGPROCESS( spLogComp	 := MSG.COMP_A5, 
									spLogAction	 := MSG.ACTION_JIGC_PICK, 
									spLogStatus	 := MSG.STATUS_RUN,
									plogFlag	 := TRUE);
						RETURN;
			END_IF
		ELSIF process_I = 1 THEN
			KR2.bOutBit[ Bit1, Bit2 ] := TRUE;
			IF KR2.bInBit[ Bit1, Bit2 ] THEN
				KR2.bOutBit[ Bit1, Bit2 ] := FALSE;
				process_I := 2;
				AUTO_MODE.processnameA5 := CONCAT(MSG.COMP_A5,MSG.ACTION_JIGC_PICK);
				AUTO_MODE.processnameA5 := CONCAT(AUTO_MODE.processnameA5,MSG.STATUS_ACK);
				LOGPROCESS( spLogComp	 := MSG.COMP_A5, 
							spLogAction	 := MSG.ACTION_JIGC_PICK, 
							spLogStatus	 := MSG.STATUS_ACK,
							plogFlag	 := TRUE);
				RETURN;
			END_IF
		ELSIF process_I = 2 THEN
			KR2.bOutBit[ Bit1, Bit2 ] := FALSE;
			IF NOT KR2.bInBit[ Bit1, Bit2 ] THEN
				process_I := 3;
				AUTO_MODE.processnameA5 := CONCAT(MSG.COMP_A5,MSG.ACTION_JIGC_PICK);
				AUTO_MODE.processnameA5 := CONCAT(AUTO_MODE.processnameA5,MSG.STATUS_DONE);
				LOGPROCESS( spLogComp	 := MSG.COMP_A5, 
							spLogAction	 := MSG.ACTION_JIGC_PICK, 
							spLogStatus	 := MSG.STATUS_DONE,
							plogFlag	 := TRUE);
				RETURN;
			END_IF
		ELSIF process_I = 3 THEN
			IF KR2.Idle THEN
				AUTO_MODE.JIGC_LOAD := FALSE;
				process_I := 4;
				A5_sequence := 16;
				AUTO_MODE.next_step := FALSE;
				AUTO_MODE.processnameA5 := CONCAT(MSG.COMP_A5,MSG.ACTION_JIGC_PICK);
				AUTO_MODE.processnameA5 := CONCAT(AUTO_MODE.processnameA5,MSG.STATUS_COMP);
				LOGPROCESS( spLogComp	 := MSG.COMP_A5, 
							spLogAction	 := MSG.ACTION_JIGC_PICK, 
							spLogStatus	 := MSG.STATUS_COMP,
							plogFlag	 := TRUE);
			END_IF
		END_IF
	
	// PLACE TO CR (KR2) ------------------------------------------------------------------------------------------
	16:
		IF process_K = 0 THEN
			SEQ_CR_PLACE();
			IF SEQ_CR_PLACE.CR_found THEN
				IF KR2.Idle AND AUTO_MODE.JIGC_PICK THEN
					CASE SEQ_CR_PLACE.CR_place_Rack OF
						1:
//							Bit1 						:= 3; 
//							Bit2 						:= 5;
							KR2.bOutBit[ Bit1, Bit2 ] 	:= TRUE;
							Msg_PlaceCR 				:= MSG.ACTION_PLACE_TO_CR1;
							process_K 					:= 1;
						2:
							Bit1 						:= 3; 
							Bit2 						:= 6;
							KR2.bOutBit[ Bit1, Bit2 ] 	:= TRUE;
							Msg_PlaceCR 				:= MSG.ACTION_PLACE_TO_CR2;
							process_K 					:= 1;
						3:
							Bit1 						:= 3; 
							Bit2 						:= 7;
							KR2.bOutBit[ Bit1, Bit2 ] 	:= TRUE;
							Msg_PlaceCR 				:= MSG.ACTION_PLACE_TO_CR3;
							process_K 					:= 1;
						4:
							Bit1 						:= 4; 
							Bit2 						:= 0;
							KR2.bOutBit[ Bit1, Bit2 ] 	:= TRUE;
							Msg_PlaceCR 				:= MSG.ACTION_PLACE_TO_CR4;
							process_K 					:= 1;
						5:
							Bit1 						:= 4; 
							Bit2 						:= 1;
							KR2.bOutBit[ Bit1, Bit2 ] 	:= TRUE;
							Msg_PlaceCR 				:= MSG.ACTION_PLACE_TO_CR5;
							process_K 					:= 1;
						6:
							Bit1 						:= 4; 
							Bit2 						:= 2;
							KR2.bOutBit[ Bit1, Bit2 ] 	:= TRUE;
							Msg_PlaceCR 				:= MSG.ACTION_PLACE_TO_CR6;
							process_K 					:= 1;
						7:
							Bit1 						:= 4; 
							Bit2 						:= 3;
							KR2.bOutBit[ Bit1, Bit2 ] 	:= TRUE;
							Msg_PlaceCR 				:= MSG.ACTION_PLACE_TO_CR7;
							process_K 					:= 1;
						8:
//							Bit1 						:= 4; 
//							Bit2 						:= 4;
							KR2.bOutBit[ Bit1, Bit2 ] 	:= TRUE;
							Msg_PlaceCR 				:= MSG.ACTION_PLACE_TO_CR8;
							process_K 					:= 1;
						9:
							Bit1 						:= 4; 
							Bit2 						:= 5;
							KR2.bOutBit[ Bit1, Bit2 ] 	:= TRUE;
							Msg_PlaceCR 				:= MSG.ACTION_PLACE_TO_CR9;
							process_K 					:= 1;
						10:
							Bit1 						:= 4; 
							Bit2 						:= 6;
							KR2.bOutBit[ Bit1, Bit2 ] 	:= TRUE;
							Msg_PlaceCR 				:= MSG.ACTION_PLACE_TO_CR10;
							process_K 					:= 1;
						11:
							Bit1 						:= 4; 
							Bit2 						:= 7;
							KR2.bOutBit[ Bit1, Bit2 ] 	:= TRUE;
							Msg_PlaceCR 				:= MSG.ACTION_PLACE_TO_CR11;
							process_K 					:= 1;
						12:
							Bit1 						:= 5; 
							Bit2 						:= 0;
							KR2.bOutBit[ Bit1, Bit2 ] 	:= TRUE;
							Msg_PlaceCR 				:= MSG.ACTION_PLACE_TO_CR12;
							process_K 					:= 1;
						13:
							Bit1 						:= 5; 
							Bit2 						:= 1;
							KR2.bOutBit[ Bit1, Bit2 ] 	:= TRUE;
							Msg_PlaceCR 				:= MSG.ACTION_PLACE_TO_CR13;
							process_K 					:= 1;
						14: 
							Msg_PlaceCR 				:= MSG.ACTION_PLACE_TO_CR14;
							process_K 					:= 1;
						15:
//							Bit1 						:= 5; 
//							Bit2 						:= 2;
							KR2.bOutBit[ Bit1, Bit2 ] 	:= TRUE;
							Msg_PlaceCR 				:= MSG.ACTION_PLACE_TO_CR15;
							process_K 					:= 1;
						16:
							Bit1 						:= 5; 
							Bit2 						:= 3;
							KR2.bOutBit[ Bit1, Bit2 ] 	:= TRUE;
							Msg_PlaceCR 				:= MSG.ACTION_PLACE_TO_CR16;
							process_K 					:= 1;
						17:
							Bit1 						:= 5; 
							Bit2 						:= 4;
							KR2.bOutBit[ Bit1, Bit2 ] 	:= TRUE;
							Msg_PlaceCR 				:= MSG.ACTION_PLACE_TO_CR17;
							process_K 					:= 1;
						18:
							Bit1 						:= 5; 
							Bit2 						:= 5;
							KR2.bOutBit[ Bit1, Bit2 ] 	:= TRUE;
							Msg_PlaceCR 				:= MSG.ACTION_PLACE_TO_CR18;
							process_K 					:= 1;
						19:
							Bit1 						:= 5; 
							Bit2 						:= 6;
							KR2.bOutBit[ Bit1, Bit2 ] 	:= TRUE;
							Msg_PlaceCR 				:= MSG.ACTION_PLACE_TO_CR19;
							process_K 					:= 1;
						20:
							Bit1 						:= 5; 
							Bit2 						:= 7;
							KR2.bOutBit[ Bit1, Bit2 ] 	:= TRUE;
							Msg_PlaceCR 				:= MSG.ACTION_PLACE_TO_CR20;
							process_K 					:= 1;
						21:
							Bit1 						:= 6; 
							Bit2 						:= 0;
							KR2.bOutBit[ Bit1, Bit2 ] 	:= TRUE;
							Msg_PlaceCR 				:= MSG.ACTION_PLACE_TO_CR21;
							process_K 					:= 1;
					END_CASE
				
					AUTO_MODE.processnameA5 := CONCAT(MSG.COMP_A5,Msg_PlaceCR);
					AUTO_MODE.processnameA5 := CONCAT(AUTO_MODE.processnameA5,MSG.STATUS_RUN);
					LOGPROCESS( spLogComp	 := MSG.COMP_A5, 
								spLogAction	 := Msg_PlaceCR, 
								spLogStatus	 := MSG.STATUS_RUN,
								plogFlag	 := TRUE);	
				END_IF
			END_IF
		ELSIF process_K = 1 THEN
			KR2.bOutBit[ Bit1, Bit2 ] := TRUE;
			IF KR2.bInBit[ Bit1, Bit2] THEN
				KR2.bOutBit[ Bit1, Bit2 ] := FALSE;
				process_K := 2;
				AUTO_MODE.processnameA5 := CONCAT(MSG.COMP_A5,MSG.ACTION_PLACE_TO_CR);
				AUTO_MODE.processnameA5 := CONCAT(AUTO_MODE.processnameA5,MSG.STATUS_ACK);
				LOGPROCESS( spLogComp	 := MSG.COMP_A5, 
							spLogAction	 := MSG.ACTION_PLACE_TO_CR, 
							spLogStatus	 := MSG.STATUS_ACK,
							plogFlag	 := TRUE);
				RETURN;
			END_IF
		ELSIF process_K = 2 THEN
			KR2.bOutBit[ Bit1, Bit2] := FALSE;
			IF NOT KR2.bInBit[ Bit1, Bit2] THEN
				process_K := 3;
				AUTO_MODE.processnameA5 := CONCAT(MSG.COMP_A5,MSG.ACTION_PLACE_TO_CR);
				AUTO_MODE.processnameA5 := CONCAT(AUTO_MODE.processnameA5,MSG.STATUS_DONE);
				LOGPROCESS( spLogComp	 := MSG.COMP_A5, 
							spLogAction	 := MSG.ACTION_PLACE_TO_CR, 
							spLogStatus	 := MSG.STATUS_DONE,
							plogFlag	 := TRUE);
				RETURN;
			END_IF
		ELSIF process_K = 3 THEN
			IF KR2.Idle THEN
				AUTO_MODE.JIGC_PICK := FALSE;
				SEQ_CR_PLACE.CR_found := FALSE;
				process_K := 4;
				A5_sequence := 17;
				AUTO_MODE.next_step := FALSE;
				AUTO_MODE.processnameA5 := CONCAT(MSG.COMP_A5,MSG.ACTION_PLACE_TO_CR);
				AUTO_MODE.processnameA5 := CONCAT(AUTO_MODE.processnameA5,MSG.STATUS_COMP);
				LOGPROCESS( spLogComp	 := MSG.COMP_A5, 
							spLogAction	 := MSG.ACTION_PLACE_TO_CR, 
							spLogStatus	 := MSG.STATUS_COMP,
							plogFlag	 := TRUE);
			END_IF
		END_IF
	// END (KR2) -------------------------------------------------------------------------------------------------------
	17:
		A5_sequence := 0;
		IF_RACK_CHECK.checkIn_A5 := FALSE;
		AUTO_MODE.next_step := FALSE;
		AUTO_MODE.processnameA5 := CONCAT(MSG.COMP_A5,MAIN.fb_TimeStamp.SystemTime);
		AUTO_MODE.processnameA5 := CONCAT(AUTO_MODE.processnameA5,MSG.STATUS_END);
		LOGPROCESS( spLogComp	 := MSG.COMP_A5, 
					spLogAction	 := MSG.ACTION_IF_TO_CR, 
					spLogStatus	 := MSG.STATUS_END,
					plogFlag	 := TRUE);
		
END_CASE

END_PROGRAM

// ---- POUs/LOGGING/LOGPROCESS.TcPOU
PROGRAM LOGPROCESS
VAR_INPUT
	spLogEvent	: STRING;
	spLogComp	: STRING;
	spLogAction	: STRING;
	spLogStatus	: STRING;
	plogFlag		: BOOL;
END_VAR
VAR_OUTPUT
	plog_complete : BOOL := FALSE;
	plog_error	 : BOOL := FALSE;
END_VAR
VAR
	fb_TimeStamp : FB_UpdateTimeStamp ();
	fbCreateDir	 : FB_CreateDir;
	fbFileOpen	 : FB_FileOpen;
	fbFileWrite	 : FB_FilePuts;
	fbFileClose	 : FB_FileClose;
	plog_state	 : ( INIT, 
					 CREATE_DIR, 
					 FILE_OPEN,
					 WRITE_TITLE,
					 WRITE_LOG, 
					 FILE_CLOSE,
					 CLEAR, 
					 ERROR);
					
	pwritepLog	 : STRING[255];
	pwriteTitle	 : STRING;
	spFolderName	 : STRING;
	spwFolderName	 : STRING;
	spFileName	 : STRING;
	spTextLog	 : STRING;
	spwTextLog	 : STRING;
	plastFileName : STRING;	
	spwLogEvent	: STRING;
	spwLogComp	: STRING;
	spwLogAction	: STRING;
	spwLogStatus	: STRING;
	
END_VAR

IF spLogComp<>spwLogComp OR spLogAction<>spwLogAction OR spLogStatus<>spwLogStatus THEN
//	spwLogEvent		:= spLogEvent;
	spwLogComp		:= spLogComp;
	spwLogAction	:= spLogAction;
	spwLogStatus	:= spLogStatus;
ELSE
	RETURN;
END_IF

spTextLog := str_concat(spwLogComp,spwLogAction,spwLogStatus);

WHILE plogFlag DO
	CASE plog_state OF
		// INIT -------------------------------------------------------------------
		INIT:
			plog_complete	:= FALSE;
			plog_error		:= FALSE;
			plog_state 		:= CREATE_DIR;
			fbCreateDir(bExecute:= FALSE);
	
		// CREATE_DIR -------------------------------------------------------------			
		CREATE_DIR:	
			spFolderName := CONCAT('C:\Users\Administrator\Desktop\log\PROCESS\', MAIN.fb_TimeStamp.SystemDate);
//			spFolderName := CONCAT('C:\Users\celli\OneDrive\Desktop\YISB_LOG\PROCESS\', MAIN.fb_TimeStamp.SystemDate);

			IF spFolderName = spwFolderName THEN
				plog_state := FILE_OPEN;
				fbCreateDir(bExecute := FALSE);
				fbFileOpen(bExecute := FALSE);
			ELSE
				fbCreateDir( sPathName:= spFolderName, bExecute:= TRUE );
				IF NOT fbCreateDir.bBusy THEN
					plog_state := FILE_OPEN;
					fbCreateDir(bExecute := FALSE);
					fbFileOpen(bExecute := FALSE);
					spwFolderName := spFolderName;
				END_IF
			END_IF
			
		// FILE_OPEN -------------------------------------------------------------
		FILE_OPEN:
			spFileName := CONCAT(spFolderName,'\');
			spFileName := CONCAT(spFileName, MAIN.fb_TimeStamp.SystemHour);
			spFileName := CONCAT(spFileName,'.csv');
				
			fbFileOpen( sPathName:= spFileName, 
						nMode:= FOPEN_MODEAPPEND, 
						bExecute:= TRUE, 
						hFile=>);
			IF fbFileOpen.bError THEN
				plog_state := ERROR;
				fbFileOpen(bExecute := FALSE);
				fbFileWrite(bExecute := FALSE);
			ELSIF NOT fbFileOpen.bBusy THEN
				plog_state := WRITE_TITLE;
				fbFileOpen(bExecute := FALSE);
				fbFileWrite(bExecute := FALSE);
			END_IF
			
		// WRITE_TITLE -------------------------------------------------------------
		WRITE_TITLE:
			IF plastFileName <> spFileName THEN	
				pwriteTitle := CONCAT('$n','Time Stamp');
				pwriteTitle := CONCAT(pwriteTitle,';');
				pwriteTitle := CONCAT(pwriteTitle,'Component');
				pwriteTitle := CONCAT(pwriteTitle,';');
				pwriteTitle := CONCAT(pwriteTitle,'Action');
				pwriteTitle := CONCAT(pwriteTitle,';');
				pwriteTitle := CONCAT(pwriteTitle,'Status');
				
				fbFileWrite ( hFile:=fbFileOpen.hFile,
								sLine:=pwriteTitle,
								bExecute:=TRUE);
				IF fbFileWrite.bError THEN
					plog_state := ERROR;
					fbFileWrite(bExecute := FALSE);
					fbFileClose(bExecute := FALSE);
				ELSIF NOT fbFileWrite.bBusy THEN
					plog_state := WRITE_LOG;
					fbFileWrite(bExecute := FALSE);
					fbFileClose(bExecute := FALSE);
					plastFileName := spFileName;
				END_IF
			ELSE
				plog_state := WRITE_LOG;
			END_IF

		// WRITE_LOG -------------------------------------------------------------
		WRITE_LOG:	
			pwritepLog := spTextLog;
			
			fbFileWrite ( hFile:=fbFileOpen.hFile,
							sLine:=pwritepLog,
							bExecute:=TRUE);
			IF fbFileWrite.bError THEN
				plog_state := ERROR;
				fbFileWrite(bExecute := FALSE);
				fbFileClose(bExecute := FALSE);
			ELSIF NOT fbFileWrite.bBusy THEN
				plog_state := FILE_CLOSE;
				fbFileWrite(bExecute := FALSE);
				fbFileClose(bExecute := FALSE);
			END_IF
			
		// FILE_CLOSE -------------------------------------------------------------
		FILE_CLOSE:			
			fbFileClose( hFile:=fbFileOpen.hFile,
						 bExecute:=TRUE);
			IF fbFileClose.bError THEN
				plog_state := ERROR;
				fbFileClose(bExecute := FALSE);
			ELSIF NOT fbFileClose.bBusy THEN
				plog_state := CLEAR;
				fbFileClose(bExecute := FALSE);
			END_IF
			
		// CLEAR -------------------------------------------------------------	
		CLEAR:
			plog_complete	:= TRUE;
			plogFlag		:= FALSE;
			plog_state 		:= INIT;
				
		// ERROR -------------------------------------------------------------	
		ERROR:
			plog_error		:= TRUE;
			plogFlag		:= FALSE;
			plog_state 		:= INIT;
	END_CASE
END_WHILE

METHOD str_concat : STRING
VAR_INPUT
	text1	: STRING;
	text2	: STRING;
	text3	: STRING;
END_VAR
VAR
	Con_String : String;
END_VAR
Con_String := CONCAT('$n', MAIN.fb_TimeStamp.FullSystemTime);
Con_String := CONCAT(Con_String, ' ; ');
Con_String := CONCAT(Con_String, text1);
Con_String := CONCAT(Con_String, ' ; ');
Con_String := CONCAT(Con_String, text2);
Con_String := CONCAT(Con_String, ' ; ');
Con_String := CONCAT(Con_String, text3);

str_concat := Con_String;
END_METHOD

END_PROGRAM

// ---- POUs/Auto_Seq/SEQ_CR_PLACE.TcPOU
PROGRAM SEQ_CR_PLACE
VAR_INPUT
	CR_Place_Rack	: UINT;
	CR_found		: BOOL;
END_VAR
VAR
	CR_place_num 	: UINT;
END_VAR

// Get next CR POS
IF NOT CR_found THEN
//	FOR CR_place_num := GVL.CR_NextPlaceNum TO 6 BY 1 DO
	FOR CR_place_num := 2 TO 21 BY 1 DO
		IF GVL.CR_NextPlaceNum > 21 OR GVL.CR_NextPlaceNum < 2 THEN
			GVL.CR_NextPlaceNum := CR_place_num := 2;
		END_IF
		IF GVL.CR_NextPlaceNum = 14 OR GVL.CR_NextPlaceNum = 8 OR GVL.CR_NextPlaceNum = 15 THEN
			GVL.CR_NextPlaceNum := GVL.CR_NextPlaceNum+1;
		ELSIF NOT COOL_RACK.CR[CR_place_num] THEN
			CR_Place_Rack		:= CR_place_num;
			GVL.CR_NextPlaceNum := CR_place_num +1 ;
			CR_found 			:= TRUE;
			RETURN;
		END_IF
	END_FOR
END_IF

END_PROGRAM

// ---- POUs/Auto_Seq/SEQ_A4.TcPOU
PROGRAM SEQ_A4
VAR_INPUT
	A4_sequence	: UINT;
	process_A	: UINT; // IF RACK PICK (KR5)
	process_J	: UINT; // PLACE TO JIG A (KR5)
	process_B	: UINT; // JIG A WELDING(KR3)
	process_C	: UINT; // JIG A TO JIG B {KR5}
	process_D	: UINT; // JIG B WELDING (KR3 KR4) 
	process_E	: UINT; // JIG B TO TWINTORCH (KR5) 
	process_F	: UINT; // TWINTORCH TO JIG C (KR5)
	process_G	: UINT; // BRACKET TO JIG C (KR2) 
	process_H	: UINT; // JIG C WELDING (KR4)
	process_I	: UINT; // JIG C TO PICK (KR2)
	process_K	: UINT; // PLACE TO CR (KR2)
	
END_VAR
VAR
	Bit1			: INT;
	Bit2			: INT;
	Jig_ErrorTime 	: TIME := T#5S;
	TT_ErrorTime 	: TIME := T#120S;
	JigTimerA 		: TON;
	JigTimerB 		: TON;
	JigTimerC 		: TON;
	TTTimer			: TON;
	Msg_PlaceCR		: STRING;
END_VAR

IF NOT IF_RACK_CHECK.checkIn_A4 
OR NOT INFEED_RACK.IFRack_Ready THEN
	RETURN;
END_IF

CASE A4_sequence OF
	// INITIATE --------------------------------------------------------------------------------------------------------------		
	0:
		process_A := 0;
		process_B := 0;
		process_C := 0;
		process_D := 0;
		process_E := 0;
		process_F := 0;
		process_G := 0;
		process_H := 0;
		process_I := 0;
		process_J := 0;
		process_K := 0;
		
		JigTimerA (IN:= FALSE);
		JigTimerB (IN:= FALSE);
		JigTimerC (IN:= FALSE);
		TTTimer	  (IN:= FALSE);
		
		AUTO_MODE.JIGA_ErrorState 	:= FALSE;
		AUTO_MODE.JIGB_ErrorState 	:= FALSE;
		AUTO_MODE.JIGC_ErrorState 	:= FALSE;
		AUTO_MODE.TT_ErrorState 	:= FALSE;
		
		AUTO_MODE.processnameA4 := CONCAT(MSG.COMP_A4,MSG.ACTION_INIT);
		LOGPROCESS( spLogComp	 := MSG.COMP_A4, 
		 			spLogAction	 := MSG.ACTION_INIT, 
		 			spLogStatus	 := MSG.STATUS_DONE,
	 	 		 	plogFlag	 := TRUE);
	
		A4_sequence := 1;
		
	// IF RACK PICK (KR5) --------------------------------------------------------------------------------------------------------------		
	1:
		IF process_A = 0 THEN
			Bit1 := 3; 
			Bit2 := 6; //205
			IF 	KR3.Idle AND 
				KR5.Idle AND 
				GVL.JIGA_Standby AND
				NOT AUTO_MODE.JIGA_LOAD AND
				NOT AUTO_MODE.IF_PICK THEN
						KR5.bOutBit[ Bit1,Bit2 ] := TRUE;
						AUTO_MODE.IF_PICK := TRUE;
						process_A := 1;
						AUTO_MODE.processnameA4 := CONCAT(MSG.COMP_A4,MSG.ACTION_IF_A4);
						AUTO_MODE.processnameA4 := CONCAT(AUTO_MODE.processnameA4,MSG.STATUS_RUN);
						LOGPROCESS( spLogComp	 := MSG.COMP_A4, 
									spLogAction	 := MSG.ACTION_IF_A4, 
									spLogStatus	 := MSG.STATUS_RUN,
									plogFlag	 := TRUE);
						RETURN;
			END_IF
		ELSIF process_A = 1 THEN
			KR5.bOutBit[ Bit1,Bit2 ] := TRUE; 
			IF KR5.bInBit[ Bit1,Bit2 ] THEN
				KR5.bOutBit[ Bit1,Bit2 ] := FALSE; 
				process_A := 2;
				AUTO_MODE.processnameA4 := CONCAT(MSG.COMP_A4,MSG.ACTION_IF_A4);
				AUTO_MODE.processnameA4 := CONCAT(AUTO_MODE.processnameA4,MSG.STATUS_ACK);
				LOGPROCESS( spLogComp	 := MSG.COMP_A4, 
							spLogAction	 := MSG.ACTION_IF_A4, 
							spLogStatus	 := MSG.STATUS_ACK,
							plogFlag	 := TRUE);
				RETURN;
			END_IF	
		ELSIF process_A = 2 THEN
			KR5.bOutBit[ Bit1,Bit2 ] := FALSE; 
			IF NOT KR5.bInBit[ Bit1,Bit2 ] THEN
				process_A:= 3;
				AUTO_MODE.processnameA4 := CONCAT(MSG.COMP_A4,MSG.ACTION_IF_A4);
				AUTO_MODE.processnameA4 := CONCAT(AUTO_MODE.processnameA4,MSG.STATUS_DONE);
				LOGPROCESS( spLogComp	 := MSG.COMP_A4, 
							spLogAction	 := MSG.ACTION_IF_A4, 
							spLogStatus	 := MSG.STATUS_DONE,
							plogFlag	 := TRUE);
				RETURN;
			END_IF	
		ELSIF process_A = 3 THEN
			IF KR5.Idle THEN
				process_A := 4;
				A4_sequence := 2;
				AUTO_MODE.next_step := FALSE;
				AUTO_MODE.processnameA4 := CONCAT(MSG.COMP_A4,MSG.ACTION_IF_A4);
				AUTO_MODE.processnameA4 := CONCAT(AUTO_MODE.processnameA4,MSG.STATUS_COMP);
				LOGPROCESS( spLogComp	 := MSG.COMP_A4, 
							spLogAction	 := MSG.ACTION_IF_A4, 
							spLogStatus	 := MSG.STATUS_COMP,
							plogFlag	 := TRUE);
			END_IF
		END_IF	
		
	// PLACE TO JIG A (KR5) --------------------------------------------------------------------------------------------------------------		
	2:
		IF process_J = 0 THEN
			Bit1 := 3; 
			Bit2 := 0; //200
			IF 	KR3.Idle AND 
				KR5.Idle AND
				GVL.JIGA_Standby AND 
				AUTO_MODE.IF_PICK AND 
				NOT AUTO_MODE.JIGA_LOAD THEN 
						KR5.bOutBit[ Bit1,Bit2 ] := TRUE;
						AUTO_MODE.JIGA_LOAD := TRUE;
						process_J := 1;
						AUTO_MODE.processnameA4 := CONCAT(MSG.COMP_A4,MSG.ACTION_JIGA_PLACE);
						AUTO_MODE.processnameA4 := CONCAT(AUTO_MODE.processnameA4,MSG.STATUS_RUN);
						LOGPROCESS( spLogComp	 := MSG.COMP_A4, 
									spLogAction	 := MSG.ACTION_JIGA_PLACE, 
									spLogStatus	 := MSG.STATUS_RUN,
									plogFlag	 := TRUE);
						RETURN;
			END_IF
		ELSIF process_J = 1 THEN
			KR5.bOutBit[ Bit1,Bit2 ] := TRUE;
			IF NOT KR5.bInBit[ Bit1,Bit2 ] THEN
				KR5.bOutBit[ Bit1,Bit2 ] := FALSE;
				process_J := 2;
				AUTO_MODE.processnameA4 := CONCAT(MSG.COMP_A4,MSG.ACTION_JIGA_PLACE);
				AUTO_MODE.processnameA4 := CONCAT(AUTO_MODE.processnameA4,MSG.STATUS_ACK);
				LOGPROCESS( spLogComp	 := MSG.COMP_A4, 
							spLogAction	 := MSG.ACTION_JIGA_PLACE, 
							spLogStatus	 := MSG.STATUS_ACK,
							plogFlag	 := TRUE);
				RETURN;
			END_IF	
		ELSIF process_J = 2 THEN
			KR5.bOutBit[ Bit1,Bit2 ] := FALSE;
			IF KR5.bInBit[ Bit1,Bit2 ] THEN
				process_J:= 3;
				AUTO_MODE.processnameA4 := CONCAT(MSG.COMP_A4,MSG.ACTION_JIGA_PLACE);
				AUTO_MODE.processnameA4 := CONCAT(AUTO_MODE.processnameA4,MSG.STATUS_DONE);
				LOGPROCESS( spLogComp	 := MSG.COMP_A4, 
							spLogAction	 := MSG.ACTION_JIGA_PLACE, 
							spLogStatus	 := MSG.STATUS_DONE,
							plogFlag	 := TRUE);
				RETURN;
			END_IF	
		ELSIF process_J = 3 THEN
			IF 	KR5.Idle AND  
				AUTO_MODE.JIGA_LOAD AND
				NOT GVL.JIGA_Standby THEN
						AUTO_MODE.IF_PICK := FALSE;
						process_J := 4;
						A4_sequence := 3;
						AUTO_MODE.next_step := FALSE;
						AUTO_MODE.processnameA4 := CONCAT(MSG.COMP_A4,MSG.ACTION_JIGA_PLACE);
						AUTO_MODE.processnameA4 := CONCAT(AUTO_MODE.processnameA4,MSG.STATUS_COMP);
						LOGPROCESS( spLogComp	 := MSG.COMP_A4, 
									spLogAction	 := MSG.ACTION_JIGA_PLACE, 
									spLogStatus	 := MSG.STATUS_COMP,
									plogFlag	 := TRUE);
			END_IF
		END_IF	
	
	// JIG A CLAMP -----------------------------------------------------------------------------------------------------------------------
	3:
		IF NOT AUTO_MODE.Halt_Production THEN
			GVL.JIGA_Clamp := TRUE;
			GVL.JIGA_Release := FALSE;
			JigTimerA(IN := TRUE, PT := JIG_ErrorTime);
		END_IF
		//insert Jig safety check here 
		
		IF JigTimerA.Q THEN
			AUTO_MODE.JIGA_ErrorState := TRUE;
			IF GVL.ClearError THEN
				JigTimerA(IN:= FALSE);
				GVL.ClearError := FALSE;
			ELSE
				AUTO_MODE.Halt_Production := TRUE;
				AUTO_MODE.processnameA4 := CONCAT(MSG.COMP_A4,MSG.ACTION_JIGA_CLAMP);
				AUTO_MODE.processnameA4 := CONCAT(AUTO_MODE.processnameA4,MSG.STATUS_ERROR);
				LOGPROCESS( spLogComp	 := MSG.COMP_A4, 
							spLogAction	 := MSG.ACTION_JIGA_CLAMP, 
							spLogStatus	 := MSG.STATUS_ERROR,
							plogFlag	 := TRUE);
			END_IF
		ELSIF GVL.JIGA_Ready THEN
			JigTimerA(IN := FALSE);
			AUTO_MODE.JIGA_ErrorState := FALSE;
			AUTO_MODE.next_step := FALSE;
			AUTO_MODE.processnameA4 := CONCAT(MSG.COMP_A4,MSG.ACTION_JIGA_CLAMP);
			AUTO_MODE.processnameA4 := CONCAT(AUTO_MODE.processnameA4,MSG.STATUS_DONE);
			LOGPROCESS( spLogComp	 := MSG.COMP_A4, 
						spLogAction	 := MSG.ACTION_JIGA_CLAMP, 
						spLogStatus	 := MSG.STATUS_COMP,
						plogFlag	 := TRUE);
			IF GVL.KR2_bypass THEN
				process_B	:= 3;	
				A4_sequence := 4;
			ELSE	
				process_B	:= 0;	
				A4_sequence := 4;
			END_IF
		END_IF
		
	// JIG A WELDING(KR3) ------------------------------------------------------------------------------------------------------------------
	4:
		IF process_B = 0 THEN
			Bit1 := 3; 
			Bit2 := 0; //300
			IF 	KR3.Idle AND 
//				KR5.Idle AND
				GVL.JIGA_Ready AND  
				NOT AUTO_MODE.JIGA_WELDING AND 
				NOT AUTO_MODE.JIGB_WELDING THEN
						KR3.bOutBit[ Bit1,Bit2 ] := TRUE;
						AUTO_MODE.JIGA_WELDING := TRUE;
						process_B := 1;
						AUTO_MODE.processnameA4 := CONCAT(MSG.COMP_A4,MSG.ACTION_JIGA_WELDING);
						AUTO_MODE.processnameA4 := CONCAT(AUTO_MODE.processnameA4,MSG.STATUS_RUN);
						LOGPROCESS( spLogComp	 := MSG.COMP_A4, 
									spLogAction	 := MSG.ACTION_JIGA_WELDING, 
									spLogStatus	 := MSG.STATUS_RUN,
									plogFlag	 := TRUE);
									RETURN;
			END_IF
		ELSIF process_B = 1 THEN 
			KR3.bOutBit[ Bit1,Bit2 ] := TRUE;
			IF NOT KR3.bInBit[ Bit1,Bit2 ] THEN
				KR3.bOutBit[ Bit1,Bit2 ] := FALSE;	
				process_B := 2;
				AUTO_MODE.processnameA4 := CONCAT(MSG.COMP_A4,MSG.ACTION_JIGA_WELDING);
				AUTO_MODE.processnameA4 := CONCAT(AUTO_MODE.processnameA4,MSG.STATUS_ACK);
				LOGPROCESS( spLogComp	 := MSG.COMP_A4, 
							spLogAction	 := MSG.ACTION_JIGA_WELDING, 
							spLogStatus	 := MSG.STATUS_ACK,
							plogFlag	 := TRUE);
				RETURN;
			END_IF
		ELSIF process_B = 2 THEN 
			KR3.bOutBit[ Bit1,Bit2 ] := FALSE;
			IF KR3.bInBit[ Bit1,Bit2 ] THEN
				process_B := 3;
				AUTO_MODE.processnameA4 := CONCAT(MSG.COMP_A4,MSG.ACTION_JIGA_WELDING);
				AUTO_MODE.processnameA4 := CONCAT(AUTO_MODE.processnameA4,MSG.STATUS_DONE);
				LOGPROCESS( spLogComp	 := MSG.COMP_A4, 
							spLogAction	 := MSG.ACTION_JIGA_WELDING, 
							spLogStatus	 := MSG.STATUS_DONE,
							plogFlag	 := TRUE);
				RETURN;
			END_IF
		ELSIF process_B = 3 THEN
			IF KR3.Idle THEN
				AUTO_MODE.JIGA_WELDING := FALSE;
				GVL.JIGA_Clamp := FALSE;
				GVL.JIGA_Release := TRUE;
				JigTimerA(IN:= FALSE);
				AUTO_MODE.processnameA4 := CONCAT(MSG.COMP_A4,MSG.ACTION_JIGA_RELEASE);
				AUTO_MODE.processnameA4 := CONCAT(AUTO_MODE.processnameA4,MSG.STATUS_DONE);
				LOGPROCESS( spLogComp	 := MSG.COMP_A4, 
							spLogAction	 := MSG.ACTION_JIGA_RELEASE, 
							spLogStatus	 := MSG.STATUS_DONE,
							plogFlag	 := TRUE);
				process_B := 4;
				AUTO_MODE.processnameA4 := CONCAT(MSG.COMP_A4,MSG.ACTION_JIGA_WELDING);
				AUTO_MODE.processnameA4 := CONCAT(AUTO_MODE.processnameA4,MSG.STATUS_COMP);
				LOGPROCESS( spLogComp	 := MSG.COMP_A4, 
							spLogAction	 := MSG.ACTION_JIGA_WELDING, 
							spLogStatus	 := MSG.STATUS_COMP,
							plogFlag	 := TRUE);
			END_IF
		ELSIF process_B = 4 THEN
			IF NOT AUTO_MODE.Halt_Production THEN
				GVL.JIGA_Clamp 		:= FALSE;
				GVL.JIGA_Release 	:= TRUE;
				JigTimerA(IN := TRUE, PT := JIG_ErrorTime);
			END_IF
			//insert Jig safety check here ------------------------------
			IF JigTimerA.Q THEN
				AUTO_MODE.JIGA_ErrorState := TRUE;
				IF GVL.ClearError THEN
					JigTimerA(IN:= FALSE);
					GVL.ClearError := FALSE;
				ELSE
					AUTO_MODE.Halt_Production := TRUE;
					AUTO_MODE.processnameA4 := CONCAT(MSG.COMP_A4,MSG.ACTION_JIGA_RELEASE);
					AUTO_MODE.processnameA4 := CONCAT(AUTO_MODE.processnameA4,MSG.STATUS_ERROR);
					LOGPROCESS( spLogComp	 := MSG.COMP_A4, 
								spLogAction	 := MSG.ACTION_JIGA_RELEASE, 
								spLogStatus	 := MSG.STATUS_ERROR,
								plogFlag	 := TRUE);
				END_IF
			ELSIF GVL.JIGA_Complete THEN
				JigTimerA(IN:= FALSE);
				AUTO_MODE.JIGA_ErrorState := FALSE;
				process_B := 5;
				A4_sequence := 5;
				AUTO_MODE.next_step := FALSE;
				AUTO_MODE.processnameA4 := CONCAT(MSG.COMP_A4,MSG.ACTION_JIGA_COMPLETE);
				AUTO_MODE.processnameA4 := CONCAT(AUTO_MODE.processnameA4,MSG.STATUS_COMP);
				LOGPROCESS( spLogComp	 := MSG.COMP_A4, 
							spLogAction	 := MSG.ACTION_JIGA_COMPLETE, 
							spLogStatus	 := MSG.STATUS_COMP,
							plogFlag	 := TRUE);
			END_IF
		END_IF
		
	// JIG A TO JIG B {KR5} -----------------------------------------------------------------------------------------------------------------
	5: 
		IF process_C = 0 THEN
			Bit1 := 3;
			Bit2 := 1; //201
			IF 	KR3.Idle AND 
				KR5.Idle AND 
				GVL.JIGB_Standby AND 
				NOT GVL.JIGA_Ready AND 
				NOT AUTO_MODE.JIGB_LOAD AND 
				NOT AUTO_MODE.JIGA_WELDING AND 
				NOT AUTO_MODE.JIGB_WELDING AND 
				NOT AUTO_MODE.JIGC_WELDING THEN
						AUTO_MODE.JIGB_LOAD := TRUE;
						KR5.bOutBit[ Bit1, Bit2 ] := TRUE;
						process_C := 1;
						AUTO_MODE.processnameA4 := CONCAT(MSG.COMP_A4,MSG.ACTION_JIGA_TO_JIGB);
						AUTO_MODE.processnameA4 := CONCAT(AUTO_MODE.processnameA4,MSG.STATUS_RUN);
						LOGPROCESS( spLogComp	 := MSG.COMP_A4, 
									spLogAction	 := MSG.ACTION_JIGA_TO_JIGB, 
									spLogStatus	 := MSG.STATUS_RUN,
									plogFlag	 := TRUE);
						RETURN;
			END_IF
		ELSIF process_C = 1 THEN 
			KR5.bOutBit [ Bit1, Bit2 ] := TRUE;
			IF KR5.bInBit[ Bit1, Bit2 ] THEN
				KR5.bOutBit[ Bit1, Bit2 ] := FALSE;
				process_C := 2;
				AUTO_MODE.processnameA4 := CONCAT(MSG.COMP_A4,MSG.ACTION_JIGA_TO_JIGB);
				AUTO_MODE.processnameA4 := CONCAT(AUTO_MODE.processnameA4,MSG.STATUS_ACK);
				LOGPROCESS( spLogComp	 := MSG.COMP_A4, 
							spLogAction	 := MSG.ACTION_JIGA_TO_JIGB, 
							spLogStatus	 := MSG.STATUS_ACK,
							plogFlag	 := TRUE);
				RETURN;
			END_IF
		ELSIF process_C = 2 THEN 
			KR5.bOutBit[ Bit1, Bit2 ] := FALSE;
			IF NOT KR5.bInBit[ Bit1, Bit2 ] THEN
				process_C := 3;
				AUTO_MODE.processnameA4 := CONCAT(MSG.COMP_A4,MSG.ACTION_JIGA_TO_JIGB);
				AUTO_MODE.processnameA4 := CONCAT(AUTO_MODE.processnameA4,MSG.STATUS_DONE);
				LOGPROCESS( spLogComp	 := MSG.COMP_A4, 
							spLogAction	 := MSG.ACTION_JIGA_TO_JIGB, 
							spLogStatus	 := MSG.STATUS_DONE,
							plogFlag	 := TRUE);
				RETURN;
			END_IF
		ELSIF process_C = 3 THEN
			IF 	KR5.Idle AND 
				NOT GVL.JIGB_Standby THEN
						AUTO_MODE.JIGA_LOAD := FALSE;
						process_C := 4;
						A4_sequence := 6;
						AUTO_MODE.next_step := FALSE;
						AUTO_MODE.processnameA4 := CONCAT(MSG.COMP_A4,MSG.ACTION_JIGA_TO_JIGB);
						AUTO_MODE.processnameA4 := CONCAT(AUTO_MODE.processnameA4,MSG.STATUS_COMP);
						LOGPROCESS( spLogComp	 := MSG.COMP_A4, 
									spLogAction	 := MSG.ACTION_JIGA_TO_JIGB, 
									spLogStatus	 := MSG.STATUS_COMP,
									plogFlag	 := TRUE);
			END_IF
		END_IF
		
	//	JIG B CLAMP	-----------------------------------------------------------------------------------------------------------------------
	6:
		IF NOT AUTO_MODE.Halt_Production THEN
			GVL.JIGB_Clamp := TRUE;
			GVL.JIGB_Release := FALSE;			
			JigTimerB(IN := TRUE, PT := JIG_ErrorTime);
		END_IF
		//insert Jig safety check here ------------------------------
		IF JigTimerB.Q THEN
			AUTO_MODE.JIGB_ErrorState := TRUE;
			IF GVL.ClearError THEN
				JigTimerB(IN:= FALSE);
				GVL.ClearError := FALSE;
			ELSE
				AUTO_MODE.Halt_Production := TRUE;
			AUTO_MODE.processnameA4 := CONCAT(MSG.COMP_A4,MSG.ACTION_JIGB_CLAMP);
			AUTO_MODE.processnameA4 := CONCAT(AUTO_MODE.processnameA4,MSG.STATUS_ERROR);
			LOGPROCESS( spLogComp	 := MSG.COMP_A4, 
						spLogAction	 := MSG.ACTION_JIGB_CLAMP, 
						spLogStatus	 := MSG.STATUS_DONE,
						plogFlag	 := TRUE);
			END_IF
		ELSIF GVL.JIGB_Ready THEN
			JigTimerB(IN:= FALSE);
			AUTO_MODE.JIGB_ErrorState := FALSE;
			AUTO_MODE.next_step := FALSE;
			AUTO_MODE.processnameA4 := CONCAT(MSG.COMP_A4,MSG.ACTION_JIGB_CLAMP);
			AUTO_MODE.processnameA4 := CONCAT(AUTO_MODE.processnameA4,MSG.STATUS_DONE);
			LOGPROCESS( spLogComp	 := MSG.COMP_A4, 
						spLogAction	 := MSG.ACTION_JIGB_CLAMP, 
						spLogStatus	 := MSG.STATUS_DONE,
						plogFlag	 := TRUE);
			IF GVL.KR2_bypass THEN
				process_D	:= 3;	
				A4_sequence := 7;
			ELSE	
				process_D	:= 0;	
				A4_sequence := 7;
			END_IF
		END_IF
		
	// JIG B WELDING (KR3) -------------------------------------------------------------------------------------------------------------	
	7:
		IF process_D = 0 THEN
			Bit1 := 3;
			Bit2 := 1; //301
			IF 	KR3.Idle AND 
				GVL.JIGB_Ready AND
				NOT AUTO_MODE.JIGA_WELDING AND 
				NOT AUTO_MODE.JIGB_WELDING THEN
						KR3.bOutBit[ Bit1, Bit2 ] := TRUE;
						AUTO_MODE.JIGB_WELDING := TRUE;
						process_D := 1;
						AUTO_MODE.processnameA4 := CONCAT(MSG.COMP_A4,MSG.ACTION_JIGB_WELDING);
						AUTO_MODE.processnameA4 := CONCAT(AUTO_MODE.processnameA4,MSG.STATUS_RUN);
						LOGPROCESS( spLogComp	 := MSG.COMP_A4, 
									spLogAction	 := MSG.ACTION_JIGB_WELDING, 
									spLogStatus	 := MSG.STATUS_RUN,
									plogFlag	 := TRUE);
				RETURN;
			END_IF
		ELSIF process_D = 1 THEN
			KR3.bOutBit[ Bit1, Bit2 ] := TRUE;
			IF KR3.bInBit[ Bit1, Bit2 ] THEN
				KR3.bOutBit[ Bit1, Bit2 ] := FALSE;
				process_D := 2;
				AUTO_MODE.processnameA4 := CONCAT(MSG.COMP_A4,MSG.ACTION_JIGB_WELDING);
				AUTO_MODE.processnameA4 := CONCAT(AUTO_MODE.processnameA4,MSG.STATUS_ACK);
				LOGPROCESS( spLogComp	 := MSG.COMP_A4, 
							spLogAction	 := MSG.ACTION_JIGB_WELDING, 
							spLogStatus	 := MSG.STATUS_ACK,
							plogFlag	 := TRUE);
				RETURN;
			END_IF
		ELSIF process_D = 2 THEN
			KR3.bOutBit[ Bit1, Bit2 ] := FALSE;
			IF NOT KR3.bInBit[ Bit1, Bit2 ] THEN
				process_D := 3;
				AUTO_MODE.Run_Next_Rack := TRUE;
				AUTO_MODE.processnameA4 := CONCAT(MSG.COMP_A4,MSG.ACTION_JIGB_WELDING);
				AUTO_MODE.processnameA4 := CONCAT(AUTO_MODE.processnameA4,MSG.STATUS_DONE);
				LOGPROCESS( spLogComp	 := MSG.COMP_A4, 
							spLogAction	 := MSG.ACTION_JIGB_WELDING, 
							spLogStatus	 := MSG.STATUS_DONE,
							plogFlag	 := TRUE);
				RETURN;
			END_IF
		ELSIF process_D = 3 THEN
			IF KR3.Idle THEN
				AUTO_MODE.JIGB_WELDING := FALSE;
				GVL.JIGB_Clamp := FALSE;
				GVL.JIGB_Release := TRUE;
				JigTimerB(IN:= FALSE);
				AUTO_MODE.processnameA4 := CONCAT(MSG.COMP_A4,MSG.ACTION_JIGB_RELEASE);
				AUTO_MODE.processnameA4 := CONCAT(AUTO_MODE.processnameA4,MSG.STATUS_DONE);
				LOGPROCESS( spLogComp	 := MSG.COMP_A4, 
							spLogAction	 := MSG.ACTION_JIGB_RELEASE, 
							spLogStatus	 := MSG.STATUS_DONE,
							plogFlag	 := TRUE);
				process_D := 4;
				AUTO_MODE.processnameA4 := CONCAT(MSG.COMP_A4,MSG.ACTION_JIGB_WELDING);
				AUTO_MODE.processnameA4 := CONCAT(AUTO_MODE.processnameA4,MSG.STATUS_COMP);
				LOGPROCESS( spLogComp	 := MSG.COMP_A4, 
							spLogAction	 := MSG.ACTION_JIGB_WELDING, 
							spLogStatus	 := MSG.STATUS_COMP,
							plogFlag	 := TRUE);
			END_IF
		ELSIF process_D = 4 THEN
			IF NOT AUTO_MODE.Halt_Production THEN
				GVL.JIGB_Clamp 		:= FALSE;
				GVL.JIGB_Release 	:= TRUE;
				JigTimerB(IN := TRUE, PT := JIG_ErrorTime);
			END_IF
			//insert Jig safety check here ------------------------------
			IF JigTimerB.Q THEN
				AUTO_MODE.JIGB_ErrorState := TRUE;
				IF GVL.ClearError THEN
					JigTimerB(IN:= FALSE);
					GVL.ClearError := FALSE;
				ELSE
					AUTO_MODE.Halt_Production := TRUE;
					AUTO_MODE.processnameA4 := CONCAT(MSG.COMP_A4,MSG.ACTION_JIGB_RELEASE);
					AUTO_MODE.processnameA4 := CONCAT(AUTO_MODE.processnameA4,MSG.STATUS_ERROR);
					LOGPROCESS( spLogComp	 := MSG.COMP_A4, 
								spLogAction	 := MSG.ACTION_JIGB_RELEASE, 
								spLogStatus	 := MSG.STATUS_ERROR,
								plogFlag	 := TRUE);
				END_IF
			ELSIF GVL.JIGB_Complete THEN
				JigTimerB(IN:= FALSE);
				AUTO_MODE.JIGB_ErrorState := FALSE;
				process_D := 5;
				A4_sequence := 8;
				AUTO_MODE.next_step := FALSE;
				AUTO_MODE.processnameA4 := CONCAT(MSG.COMP_A4,MSG.ACTION_JIGB_COMPLETE);
				AUTO_MODE.processnameA4 := CONCAT(AUTO_MODE.processnameA4,MSG.STATUS_COMP);
				LOGPROCESS( spLogComp	 := MSG.COMP_A4, 
							spLogAction	 := MSG.ACTION_JIGB_COMPLETE, 
							spLogStatus	 := MSG.STATUS_COMP,
							plogFlag	 := TRUE);
			END_IF
		END_IF
		
	// JIG B TO TWINTORCH (KR5) -------------------------------------------------------------------------------------------------------------
	8: 
		IF process_E = 0 THEN
			Bit1 := 3;
			Bit2 := 2; //302
//			IF 	KR3.Idle AND 
			IF	KR5.Idle AND
				GVL.TTorch_Standy AND 
				NOT AUTO_MODE.IF_PICK AND
				NOT AUTO_MODE.IF_PICK AND
				NOT AUTO_MODE.TT_LOAD AND 
				NOT GVL.JIGB_Ready AND
				NOT AUTO_MODE.JIGA_WELDING AND 
				NOT AUTO_MODE.JIGB_WELDING AND 
				NOT AUTO_MODE.TT_WELDING THEN
						AUTO_MODE.TT_LOAD := TRUE;
						KR5.bOutBit[ Bit1, Bit2 ] := TRUE;
						process_E := 1;
						AUTO_MODE.processnameA4 := CONCAT(MSG.COMP_A4,MSG.ACTION_JIGB_TO_TT);
						AUTO_MODE.processnameA4 := CONCAT(AUTO_MODE.processnameA4,MSG.STATUS_RUN);
						LOGPROCESS( spLogComp	 := MSG.COMP_A4, 
									spLogAction	 := MSG.ACTION_JIGB_TO_TT, 
									spLogStatus	 := MSG.STATUS_RUN,
									plogFlag	 := TRUE);
						RETURN;
			END_IF
		ELSIF process_E = 1 THEN
			KR5.bOutBit[ Bit1, Bit2 ] := TRUE;
			IF KR5.bInBit[ Bit1, Bit2 ] THEN
				KR5.bOutBit[ Bit1, Bit2 ] := FALSE;
				process_E := 2;
				AUTO_MODE.processnameA4 := CONCAT(MSG.COMP_A4,MSG.ACTION_JIGB_TO_TT);
				AUTO_MODE.processnameA4 := CONCAT(AUTO_MODE.processnameA4,MSG.STATUS_ACK);
				LOGPROCESS( spLogComp	 := MSG.COMP_A4, 
							spLogAction	 := MSG.ACTION_JIGB_TO_TT, 
							spLogStatus	 := MSG.STATUS_ACK,
							plogFlag	 := TRUE);
				RETURN;
			END_IF
		ELSIF process_E = 2 THEN
			KR5.bOutBit[ Bit1, Bit2 ] := FALSE;
			IF NOT KR5.bInBit[ Bit1, Bit2 ] THEN
				process_E := 3;
				AUTO_MODE.processnameA4 := CONCAT(MSG.COMP_A4,MSG.ACTION_JIGB_TO_TT);
				AUTO_MODE.processnameA4 := CONCAT(AUTO_MODE.processnameA4,MSG.STATUS_DONE);
				LOGPROCESS( spLogComp	 := MSG.COMP_A4, 
							spLogAction	 := MSG.ACTION_JIGB_TO_TT, 
							spLogStatus	 := MSG.STATUS_DONE,
							plogFlag	 := TRUE);
				RETURN;
			END_IF
		ELSIF process_E = 3 THEN
			IF KR5.Idle THEN
				AUTO_MODE.JIGB_LOAD := FALSE;
				process_E := 4;
				A4_sequence := 9;
				AUTO_MODE.next_step := FALSE;
//				AUTO_MODE.Run_Next_Rack :=TRUE;
				AUTO_MODE.processnameA4 := CONCAT(MSG.COMP_A4,MSG.ACTION_JIGB_TO_TT);
				AUTO_MODE.processnameA4 := CONCAT(AUTO_MODE.processnameA4,MSG.STATUS_COMP);
				LOGPROCESS( spLogComp	 := MSG.COMP_A4, 
							spLogAction	 := MSG.ACTION_JIGB_TO_TT, 
							spLogStatus	 := MSG.STATUS_COMP,
							plogFlag	 := TRUE);
			END_IF
		END_IF	
	
	// TWINTORCH WELDING -------------------------------------------------------------------------------------------------------------	
	9:
		//insert Jig safety check here ------------------------------
		IF NOT GVL.TTorch_Standy THEN
			GVL.TTorch_Run := TRUE;
			AUTO_MODE.TT_WELDING := TRUE;
			A4_sequence := 10;
			TTTimer(IN := TRUE, PT := TT_ErrorTime);
			AUTO_MODE.processnameA4 := CONCAT(MSG.COMP_A4,MSG.ACTION_TT_RUN);
			AUTO_MODE.processnameA4 := CONCAT(AUTO_MODE.processnameA4,MSG.STATUS_RUN);
			LOGPROCESS( spLogComp	 := MSG.COMP_A4, 
						spLogAction	 := MSG.ACTION_TT_RUN, 
						spLogStatus	 := MSG.STATUS_RUN,
						plogFlag	 := TRUE);
			RETURN;
		END_IF
	// TWINTORCH WELD COMPLETE -------------------------------------------------------------------------------------------------------------		
	10:
		
		//insert Jig safety check here ------------------------------
		IF TTTimer.Q THEN
			AUTO_MODE.TT_ErrorState := TRUE;
			IF GVL.ClearError THEN
				TTTimer(IN:= FALSE);
				GVL.ClearError := FALSE;
			ELSE
				AUTO_MODE.Halt_Production := TRUE;
				AUTO_MODE.processnameA4 := CONCAT(MSG.COMP_A4,MSG.ACTION_TT_RUN);
				AUTO_MODE.processnameA4 := CONCAT(AUTO_MODE.processnameA4,MSG.STATUS_ERROR);
				LOGPROCESS( spLogComp	 := MSG.COMP_A4, 
							spLogAction	 := MSG.ACTION_TT_RUN, 
							spLogStatus	 := MSG.STATUS_ERROR,
							plogFlag	 := TRUE);
			END_IF
		ELSIF GVL.TTorch_Complete THEN
			TTTimer(IN:= FALSE);
			AUTO_MODE.TT_ErrorState := FALSE;
			GVL.TTorch_Run := FALSE;
			AUTO_MODE.TT_WELDING := FALSE;
			A4_sequence := 11;
			AUTO_MODE.next_step := FALSE;
			AUTO_MODE.processnameA4 := CONCAT(MSG.COMP_A4,MSG.ACTION_TT_RUN);
			AUTO_MODE.processnameA4 := CONCAT(AUTO_MODE.processnameA4,MSG.STATUS_DONE);
			LOGPROCESS( spLogComp	 := MSG.COMP_A4, 
						spLogAction	 := MSG.ACTION_TT_RUN, 
						spLogStatus	 := MSG.STATUS_DONE,
						plogFlag	 := TRUE);
			RETURN;
		END_IF
		
